// TIA Portal V15.1 export
// export: Created 2024-05-17T05:38:36.3165003Z, ExportSetting WithDefaults, DisplayName Totally Integrated Automation Portal, DisplayVersion V15.1 Update 5, DisplayName TIA Portal Openness, DisplayVersion V15.1 Update 5, DisplayName SINAMICS Startdrive Advanced, DisplayVersion V15.1, DisplayName G130, G150, S120, S150, SINAMICS MV, S210, DisplayVersion V15.1, DisplayName G110M, G120, G120C, G120D, G120P, DisplayVersion V15.1, DisplayName STEP 7 Professional, DisplayVersion V15.1 Update 5, DisplayName STEP 7 Safety, DisplayVersion V15.1, DisplayName WinCC Professional, DisplayVersion V15.1 Update 5, DisplayName SIMATIC Visualization Architect, DisplayVersion V15.1
FUNCTION_BLOCK "LProcPAC-Driver"   // FB1741, SCL
TITLE = LProcPAC-Driver
{ S7_Optimized_Access := 'FALSE' }
AUTHOR : CSTAAL
VERSION : 2.0
// stored: AutoNumber false, IsIECCheckEnabled false, SetENOAutomatically False, UDAEnableTagReadback false
   VAR_INPUT
      ID { ExternalAccessible := 'False'; ExternalVisible := 'False'; ExternalWritable := 'False'} : HW_IO := 0;   // PROFINET = The diagnostic address of the SENTRON PAC; PROFIBUS = The number of the first byte of the input data of the PAC.
      First_Byte_I_O_Data { ExternalAccessible := 'False'; ExternalVisible := 'False'; ExternalWritable := 'False'} : Int := 0;   // The number of the first byte of the control bytes of the SENTRON PAC.
      Connection_Type { ExternalAccessible := 'False'; ExternalVisible := 'False'; ExternalWritable := 'False'} : Int := 1;   // The connection type of the Energy Meter: 1 = single phase, 3 = 3 phase
      Comm_Resource_Limit { ExternalAccessible := 'False'; ExternalVisible := 'False'; ExternalWritable := 'False'} : Int := 4;   // The limit of resources, which can be used by the drviers.
      Automatic_Update { ExternalAccessible := 'False'; ExternalVisible := 'False'; ExternalWritable := 'False'} : Bool := FALSE;   // TRUE = Always update the measurement values as fast as possible.
      Reset_Min_Max { ExternalAccessible := 'False'; ExternalVisible := 'False'; ExternalWritable := 'False'} : Bool := FALSE;   // FALSE ==> TRUE = Reset the minimum and maximum values.
      Reset_Energy_Counter { ExternalAccessible := 'False'; ExternalVisible := 'False'; ExternalWritable := 'False'} : Bool := FALSE;   // FALSE ==> TRUE = Reset the energy counter of the Energy Meter.
      HMI_Bits_Connected { ExternalAccessible := 'False'; ExternalVisible := 'False'; ExternalWritable := 'False'} : Bool := FALSE;   // TRUE = Structure HMI_Bits is connected; FALSE = Structure HMI_Bits is not connected
      Comm_Type { ExternalAccessible := 'False'; ExternalVisible := 'False'; ExternalWritable := 'False'} : Int := 1;   // The communication type, to the SENTRON PAC: 1 = PROFINET, 2 = PROFIBUS
      Min_Max_Calculated { ExternalAccessible := 'False'; ExternalVisible := 'False'; ExternalWritable := 'False'} : Bool := TRUE;   // Only used for PROFIBUS: TRUE = Min-Max-Values are calculated in the driver; FALSE = Min-Max-Values read from the driver.
   END_VAR
   VAR_OUTPUT
      Driver_Control { ExternalAccessible := 'False'; ExternalVisible := 'False'; ExternalWritable := 'False'} : Word;   // Driver Control
      Driver_Data { ExternalAccessible := 'False'; ExternalVisible := 'False'; ExternalWritable := 'False'} : Struct   // The structure including all measurement values. Used for the visualization and the connection to the E2M_Visu block.
         U_L1_L2 { ExternalAccessible := 'False'; ExternalVisible := 'False'; ExternalWritable := 'False'} : Real;
         U_L2_L3 { ExternalAccessible := 'False'; ExternalVisible := 'False'; ExternalWritable := 'False'} : Real;
         U_L3_L1 { ExternalAccessible := 'False'; ExternalVisible := 'False'; ExternalWritable := 'False'} : Real;
         U_L1 { ExternalAccessible := 'False'; ExternalVisible := 'False'; ExternalWritable := 'False'} : Real;
         U_L2 { ExternalAccessible := 'False'; ExternalVisible := 'False'; ExternalWritable := 'False'} : Real;
         U_L3 { ExternalAccessible := 'False'; ExternalVisible := 'False'; ExternalWritable := 'False'} : Real;
         U_L1_L2_min { ExternalAccessible := 'False'; ExternalVisible := 'False'; ExternalWritable := 'False'} : Real;
         U_L2_L3_min { ExternalAccessible := 'False'; ExternalVisible := 'False'; ExternalWritable := 'False'} : Real;
         U_L3_L1_min { ExternalAccessible := 'False'; ExternalVisible := 'False'; ExternalWritable := 'False'} : Real;
         U_L1_min { ExternalAccessible := 'False'; ExternalVisible := 'False'; ExternalWritable := 'False'} : Real;
         U_L2_min { ExternalAccessible := 'False'; ExternalVisible := 'False'; ExternalWritable := 'False'} : Real;
         U_L3_min { ExternalAccessible := 'False'; ExternalVisible := 'False'; ExternalWritable := 'False'} : Real;
         U_L1_L2_max { ExternalAccessible := 'False'; ExternalVisible := 'False'; ExternalWritable := 'False'} : Real;
         U_L2_L3_max { ExternalAccessible := 'False'; ExternalVisible := 'False'; ExternalWritable := 'False'} : Real;
         U_L3_L1_max { ExternalAccessible := 'False'; ExternalVisible := 'False'; ExternalWritable := 'False'} : Real;
         U_L1_max { ExternalAccessible := 'False'; ExternalVisible := 'False'; ExternalWritable := 'False'} : Real;
         U_L2_max { ExternalAccessible := 'False'; ExternalVisible := 'False'; ExternalWritable := 'False'} : Real;
         U_L3_max { ExternalAccessible := 'False'; ExternalVisible := 'False'; ExternalWritable := 'False'} : Real;
         U_PH_PH_Average { ExternalAccessible := 'False'; ExternalVisible := 'False'; ExternalWritable := 'False'} : Real;
         U_PH_N_Average { ExternalAccessible := 'False'; ExternalVisible := 'False'; ExternalWritable := 'False'} : Real;
         U_PH_PH_Average_min { ExternalAccessible := 'False'; ExternalVisible := 'False'; ExternalWritable := 'False'} : Real;
         U_PH_N_Average_min { ExternalAccessible := 'False'; ExternalVisible := 'False'; ExternalWritable := 'False'} : Real;
         U_PH_PH_Average_max { ExternalAccessible := 'False'; ExternalVisible := 'False'; ExternalWritable := 'False'} : Real;
         U_PH_N_Average_max { ExternalAccessible := 'False'; ExternalVisible := 'False'; ExternalWritable := 'False'} : Real;
         I_L1 { ExternalAccessible := 'False'; ExternalVisible := 'False'; ExternalWritable := 'False'} : Real;
         I_L2 { ExternalAccessible := 'False'; ExternalVisible := 'False'; ExternalWritable := 'False'} : Real;
         I_L3 { ExternalAccessible := 'False'; ExternalVisible := 'False'; ExternalWritable := 'False'} : Real;
         I_L1_min { ExternalAccessible := 'False'; ExternalVisible := 'False'; ExternalWritable := 'False'} : Real;
         I_L2_min { ExternalAccessible := 'False'; ExternalVisible := 'False'; ExternalWritable := 'False'} : Real;
         I_L3_min { ExternalAccessible := 'False'; ExternalVisible := 'False'; ExternalWritable := 'False'} : Real;
         I_L1_max { ExternalAccessible := 'False'; ExternalVisible := 'False'; ExternalWritable := 'False'} : Real;
         I_L2_max { ExternalAccessible := 'False'; ExternalVisible := 'False'; ExternalWritable := 'False'} : Real;
         I_L3_max { ExternalAccessible := 'False'; ExternalVisible := 'False'; ExternalWritable := 'False'} : Real;
         I_Average { ExternalAccessible := 'False'; ExternalVisible := 'False'; ExternalWritable := 'False'} : Real;
         I_Average_min { ExternalAccessible := 'False'; ExternalVisible := 'False'; ExternalWritable := 'False'} : Real;
         I_Average_max { ExternalAccessible := 'False'; ExternalVisible := 'False'; ExternalWritable := 'False'} : Real;
         f { ExternalAccessible := 'False'; ExternalVisible := 'False'; ExternalWritable := 'False'} : Real;
         f_min { ExternalAccessible := 'False'; ExternalVisible := 'False'; ExternalWritable := 'False'} : Real;
         f_max { ExternalAccessible := 'False'; ExternalVisible := 'False'; ExternalWritable := 'False'} : Real;
         S_Total { ExternalAccessible := 'False'; ExternalVisible := 'False'; ExternalWritable := 'False'} : Real;
         S_Total_min { ExternalAccessible := 'False'; ExternalVisible := 'False'; ExternalWritable := 'False'} : Real;
         S_Total_max { ExternalAccessible := 'False'; ExternalVisible := 'False'; ExternalWritable := 'False'} : Real;
         P_Total { ExternalAccessible := 'False'; ExternalVisible := 'False'; ExternalWritable := 'False'} : Real;
         P_Total_min { ExternalAccessible := 'False'; ExternalVisible := 'False'; ExternalWritable := 'False'} : Real;
         P_Total_max { ExternalAccessible := 'False'; ExternalVisible := 'False'; ExternalWritable := 'False'} : Real;
         Q_Total { ExternalAccessible := 'False'; ExternalVisible := 'False'; ExternalWritable := 'False'} : Real;
         Q_Total_min { ExternalAccessible := 'False'; ExternalVisible := 'False'; ExternalWritable := 'False'} : Real;
         Q_Total_max { ExternalAccessible := 'False'; ExternalVisible := 'False'; ExternalWritable := 'False'} : Real;
         Cos_L1 { ExternalAccessible := 'False'; ExternalVisible := 'False'; ExternalWritable := 'False'} : Real;
         Cos_L1_min { ExternalAccessible := 'False'; ExternalVisible := 'False'; ExternalWritable := 'False'} : Real;
         Cos_L1_max { ExternalAccessible := 'False'; ExternalVisible := 'False'; ExternalWritable := 'False'} : Real;
         Cos_L2 { ExternalAccessible := 'False'; ExternalVisible := 'False'; ExternalWritable := 'False'} : Real;
         Cos_L2_min { ExternalAccessible := 'False'; ExternalVisible := 'False'; ExternalWritable := 'False'} : Real;
         Cos_L2_max { ExternalAccessible := 'False'; ExternalVisible := 'False'; ExternalWritable := 'False'} : Real;
         Cos_L3 { ExternalAccessible := 'False'; ExternalVisible := 'False'; ExternalWritable := 'False'} : Real;
         Cos_L3_min { ExternalAccessible := 'False'; ExternalVisible := 'False'; ExternalWritable := 'False'} : Real;
         Cos_L3_max { ExternalAccessible := 'False'; ExternalVisible := 'False'; ExternalWritable := 'False'} : Real;
         Cos_Total { ExternalAccessible := 'False'; ExternalVisible := 'False'; ExternalWritable := 'False'} : Real;
         Cos_Total_min { ExternalAccessible := 'False'; ExternalVisible := 'False'; ExternalWritable := 'False'} : Real;
         Cos_Total_max { ExternalAccessible := 'False'; ExternalVisible := 'False'; ExternalWritable := 'False'} : Real;
         S_L1 { ExternalAccessible := 'False'; ExternalVisible := 'False'; ExternalWritable := 'False'} : Real;
         S_L2 { ExternalAccessible := 'False'; ExternalVisible := 'False'; ExternalWritable := 'False'} : Real;
         S_L3 { ExternalAccessible := 'False'; ExternalVisible := 'False'; ExternalWritable := 'False'} : Real;
         S_L1_min { ExternalAccessible := 'False'; ExternalVisible := 'False'; ExternalWritable := 'False'} : Real;
         S_L2_min { ExternalAccessible := 'False'; ExternalVisible := 'False'; ExternalWritable := 'False'} : Real;
         S_L3_min { ExternalAccessible := 'False'; ExternalVisible := 'False'; ExternalWritable := 'False'} : Real;
         S_L1_max { ExternalAccessible := 'False'; ExternalVisible := 'False'; ExternalWritable := 'False'} : Real;
         S_L2_max { ExternalAccessible := 'False'; ExternalVisible := 'False'; ExternalWritable := 'False'} : Real;
         S_L3_max { ExternalAccessible := 'False'; ExternalVisible := 'False'; ExternalWritable := 'False'} : Real;
         P_L1 { ExternalAccessible := 'False'; ExternalVisible := 'False'; ExternalWritable := 'False'} : Real;
         P_L2 { ExternalAccessible := 'False'; ExternalVisible := 'False'; ExternalWritable := 'False'} : Real;
         P_L3 { ExternalAccessible := 'False'; ExternalVisible := 'False'; ExternalWritable := 'False'} : Real;
         P_L1_min { ExternalAccessible := 'False'; ExternalVisible := 'False'; ExternalWritable := 'False'} : Real;
         P_L2_min { ExternalAccessible := 'False'; ExternalVisible := 'False'; ExternalWritable := 'False'} : Real;
         P_L3_min { ExternalAccessible := 'False'; ExternalVisible := 'False'; ExternalWritable := 'False'} : Real;
         P_L1_max { ExternalAccessible := 'False'; ExternalVisible := 'False'; ExternalWritable := 'False'} : Real;
         P_L2_max { ExternalAccessible := 'False'; ExternalVisible := 'False'; ExternalWritable := 'False'} : Real;
         P_L3_max { ExternalAccessible := 'False'; ExternalVisible := 'False'; ExternalWritable := 'False'} : Real;
         Q_L1 { ExternalAccessible := 'False'; ExternalVisible := 'False'; ExternalWritable := 'False'} : Real;
         Q_L2 { ExternalAccessible := 'False'; ExternalVisible := 'False'; ExternalWritable := 'False'} : Real;
         Q_L3 { ExternalAccessible := 'False'; ExternalVisible := 'False'; ExternalWritable := 'False'} : Real;
         Q_L1_min { ExternalAccessible := 'False'; ExternalVisible := 'False'; ExternalWritable := 'False'} : Real;
         Q_L2_min { ExternalAccessible := 'False'; ExternalVisible := 'False'; ExternalWritable := 'False'} : Real;
         Q_L3_min { ExternalAccessible := 'False'; ExternalVisible := 'False'; ExternalWritable := 'False'} : Real;
         Q_L1_max { ExternalAccessible := 'False'; ExternalVisible := 'False'; ExternalWritable := 'False'} : Real;
         Q_L2_max { ExternalAccessible := 'False'; ExternalVisible := 'False'; ExternalWritable := 'False'} : Real;
         Q_L3_max { ExternalAccessible := 'False'; ExternalVisible := 'False'; ExternalWritable := 'False'} : Real;
         E_Active_Rate1_Import { ExternalAccessible := 'False'; ExternalVisible := 'False'; ExternalWritable := 'False'} : Real;
         E_Active_Rate2_Import { ExternalAccessible := 'False'; ExternalVisible := 'False'; ExternalWritable := 'False'} : Real;
         E_Active_Rate1_Export { ExternalAccessible := 'False'; ExternalVisible := 'False'; ExternalWritable := 'False'} : Real;
         E_Active_Rate2_Export { ExternalAccessible := 'False'; ExternalVisible := 'False'; ExternalWritable := 'False'} : Real;
         E_Reactive_Rate1_Import { ExternalAccessible := 'False'; ExternalVisible := 'False'; ExternalWritable := 'False'} : Real;
         E_Reactive_Rate2_Import { ExternalAccessible := 'False'; ExternalVisible := 'False'; ExternalWritable := 'False'} : Real;
         E_Reactive_Rate1_Export { ExternalAccessible := 'False'; ExternalVisible := 'False'; ExternalWritable := 'False'} : Real;
         E_Reactive_Rate2_Export { ExternalAccessible := 'False'; ExternalVisible := 'False'; ExternalWritable := 'False'} : Real;
         E_Apparent_Rate1_Import { ExternalAccessible := 'False'; ExternalVisible := 'False'; ExternalWritable := 'False'} : Real;
         E_Apparent_Rate2_Import { ExternalAccessible := 'False'; ExternalVisible := 'False'; ExternalWritable := 'False'} : Real;
         RTime_Data_Energy { ExternalAccessible := 'False'; ExternalVisible := 'False'; ExternalWritable := 'False'} : Date_And_Time;
         RTime_Data_Value { ExternalAccessible := 'False'; ExternalVisible := 'False'; ExternalWritable := 'False'} : Date_And_Time;
         U_PH_PH_Mod { ExternalAccessible := 'False'; ExternalVisible := 'False'; ExternalWritable := 'False'} : Word;
         U_PH_N_Mod { ExternalAccessible := 'False'; ExternalVisible := 'False'; ExternalWritable := 'False'} : Word;
         I_Mod { ExternalAccessible := 'False'; ExternalVisible := 'False'; ExternalWritable := 'False'} : Word;
         S_Mod { ExternalAccessible := 'False'; ExternalVisible := 'False'; ExternalWritable := 'False'} : Word;
         P_Mod { ExternalAccessible := 'False'; ExternalVisible := 'False'; ExternalWritable := 'False'} : Word;
         Q_Mod { ExternalAccessible := 'False'; ExternalVisible := 'False'; ExternalWritable := 'False'} : Word;
         E_Mod { ExternalAccessible := 'False'; ExternalVisible := 'False'; ExternalWritable := 'False'} : Word;
         f_Mod { ExternalAccessible := 'False'; ExternalVisible := 'False'; ExternalWritable := 'False'} : Word;
         Cos_Mod { ExternalAccessible := 'False'; ExternalVisible := 'False'; ExternalWritable := 'False'} : Word;
         Calculate_Value1 { ExternalAccessible := 'False'; ExternalVisible := 'False'; ExternalWritable := 'False'} : Word;
         Calculate_Value2 { ExternalAccessible := 'False'; ExternalVisible := 'False'; ExternalWritable := 'False'} : Word;
         Calculate_Value3 { ExternalAccessible := 'False'; ExternalVisible := 'False'; ExternalWritable := 'False'} : Word;
         Calculate_Value4 { ExternalAccessible := 'False'; ExternalVisible := 'False'; ExternalWritable := 'False'} : Word;
         Calculate_Value5 { ExternalAccessible := 'False'; ExternalVisible := 'False'; ExternalWritable := 'False'} : Word;
         Calculate_Value6 { ExternalAccessible := 'False'; ExternalVisible := 'False'; ExternalWritable := 'False'} : Word;
         Energy_Meter_Unit { ExternalAccessible := 'False'; ExternalVisible := 'False'; ExternalWritable := 'False'} : Word;
         Rest_Start_Auto { ExternalAccessible := 'False'; ExternalVisible := 'False'; ExternalWritable := 'False'} : Bool;
         Read_Value { ExternalAccessible := 'False'; ExternalVisible := 'False'; ExternalWritable := 'False'} : Bool;
         Connection_Type { ExternalAccessible := 'False'; ExternalVisible := 'False'; ExternalWritable := 'False'} : Int;
         Driver_Error { ExternalAccessible := 'False'; ExternalVisible := 'False'; ExternalWritable := 'False'} : Int;
      END_STRUCT;
      Energy_Counter { ExternalAccessible := 'False'; ExternalVisible := 'False'; ExternalWritable := 'False'} : Struct   // The structure with all energy counter as 64-Bit float values.
         Active_Rate1_Imp_Raw { ExternalAccessible := 'False'; ExternalVisible := 'False'; ExternalWritable := 'False'} : DInt;
         Active_Rate1_Imp_Fine { ExternalAccessible := 'False'; ExternalVisible := 'False'; ExternalWritable := 'False'} : DInt;
         Active_Rate1_Exp_Raw { ExternalAccessible := 'False'; ExternalVisible := 'False'; ExternalWritable := 'False'} : DInt;
         Active_Rate1_Exp_Fine { ExternalAccessible := 'False'; ExternalVisible := 'False'; ExternalWritable := 'False'} : DInt;
         Active_Rate2_Imp_Raw { ExternalAccessible := 'False'; ExternalVisible := 'False'; ExternalWritable := 'False'} : DInt;
         Active_Rate2_Imp_Fine { ExternalAccessible := 'False'; ExternalVisible := 'False'; ExternalWritable := 'False'} : DInt;
         Active_Rate2_Exp_Raw { ExternalAccessible := 'False'; ExternalVisible := 'False'; ExternalWritable := 'False'} : DInt;
         Active_Rate2_Exp_Fine { ExternalAccessible := 'False'; ExternalVisible := 'False'; ExternalWritable := 'False'} : DInt;
         Reactive_Rate1_Imp_Raw { ExternalAccessible := 'False'; ExternalVisible := 'False'; ExternalWritable := 'False'} : DInt;
         Reactive_Rate1_Imp_Fine { ExternalAccessible := 'False'; ExternalVisible := 'False'; ExternalWritable := 'False'} : DInt;
         Reactive_Rate1_Exp_Raw { ExternalAccessible := 'False'; ExternalVisible := 'False'; ExternalWritable := 'False'} : DInt;
         Reactive_Rate1_Exp_Fine { ExternalAccessible := 'False'; ExternalVisible := 'False'; ExternalWritable := 'False'} : DInt;
         Reactive_Rate2_Imp_Raw { ExternalAccessible := 'False'; ExternalVisible := 'False'; ExternalWritable := 'False'} : DInt;
         Reactive_Rate2_Imp_Fine { ExternalAccessible := 'False'; ExternalVisible := 'False'; ExternalWritable := 'False'} : DInt;
         Reactive_Rate2_Exp_Raw { ExternalAccessible := 'False'; ExternalVisible := 'False'; ExternalWritable := 'False'} : DInt;
         Reactive_Rate2_Exp_Fine { ExternalAccessible := 'False'; ExternalVisible := 'False'; ExternalWritable := 'False'} : DInt;
         Apparent_Rate1_Imp_Raw { ExternalAccessible := 'False'; ExternalVisible := 'False'; ExternalWritable := 'False'} : DInt;
         Apparent_Rate1_Imp_Fine { ExternalAccessible := 'False'; ExternalVisible := 'False'; ExternalWritable := 'False'} : DInt;
         Apparent_Rate2_Imp_Raw { ExternalAccessible := 'False'; ExternalVisible := 'False'; ExternalWritable := 'False'} : DInt;
         Apparent_Rate2_Imp_Fine { ExternalAccessible := 'False'; ExternalVisible := 'False'; ExternalWritable := 'False'} : DInt;
      END_STRUCT;
      Time_Between_Update { ExternalAccessible := 'False'; ExternalVisible := 'False'; ExternalWritable := 'False'} : Time := T#0MS;   // The time between the current and the last update of the measurement values.
      Time_Between_Update_Max { ExternalAccessible := 'False'; ExternalVisible := 'False'; ExternalWritable := 'False'} : Time := T#0MS;   // The maximum time between two measurement value updates.
      Time_Stamp_Meas_Values { ExternalAccessible := 'False'; ExternalVisible := 'False'; ExternalWritable := 'False'} : Date_And_Time := DT#1990-01-01-00:00:00;   // The time stamp of the currently available measurement values.
      Error_Location { ExternalAccessible := 'False'; ExternalVisible := 'False'; ExternalWritable := 'False'} : Word := WORD#16#0000;   // The error location or the status of the block. Detailed information in the manual.
      Error_Code { ExternalAccessible := 'False'; ExternalVisible := 'False'; ExternalWritable := 'False'} : DWord := DWORD#16#0000_0000;   // The error code in case of an error of the block, otherwise 0. Detailed information in the manual.
   END_VAR
   VAR_IN_OUT
      HMI_Bits : Struct   // The structure with the feedback of the HMI. Used for the visualization and the connection to the E2M_Visu block.
         Start_Acyclic : Bool;
         Start_Auto : Bool;
         Reset_min_max_Data : Bool;
         Reset_Energy_Meter : Bool;
      END_STRUCT;
      Comm_Resource_Counter { ExternalAccessible := 'False'; ExternalVisible := 'False'; ExternalWritable := 'False'} : Int := 0;   // The counter of the currently used resources from all E2M drivers.
   END_VAR
   VAR
      Read_Data_Record { ExternalAccessible := 'False'; ExternalVisible := 'False'; ExternalWritable := 'False'; S7_SetPoint := 'True'} : RDREC;
      Write_Data_Record { ExternalAccessible := 'False'; ExternalVisible := 'False'; ExternalWritable := 'False'; S7_SetPoint := 'True'} : WRREC;
   END_VAR
   VAR DB_SPECIFIC
      Time_Measurement { ExternalAccessible := 'False'; ExternalVisible := 'False'; ExternalWritable := 'False'; S7_SetPoint := 'True'} : TON_TIME;
      Error_Retry_Timer { ExternalAccessible := 'False'; ExternalVisible := 'False'; ExternalWritable := 'False'; S7_SetPoint := 'True'} : TON_TIME;
      Watchdog { ExternalAccessible := 'False'; ExternalVisible := 'False'; ExternalWritable := 'False'; S7_SetPoint := 'True'} : TON_TIME;
      Reset_Timer { ExternalAccessible := 'False'; ExternalVisible := 'False'; ExternalWritable := 'False'; S7_SetPoint := 'True'} : TON_TIME;
   END_VAR
   VAR
      LREAL_TO_DINT { ExternalAccessible := 'False'; ExternalVisible := 'False'; ExternalWritable := 'False'; S7_SetPoint := 'True'} : "LProcPAC-Conversion";
   END_VAR
   VAR DB_SPECIFIC
      Input_Variables_OK { ExternalAccessible := 'False'; ExternalVisible := 'False'; ExternalWritable := 'False'} : Bool := FALSE;
      HMI_Input_Bits_Connected { ExternalAccessible := 'False'; ExternalVisible := 'False'; ExternalWritable := 'False'} : Bool := FALSE;
      Reset_En_Count_Request { ExternalAccessible := 'False'; ExternalVisible := 'False'; ExternalWritable := 'False'} : Bool := FALSE;
      Reset_Min_Max_Request { ExternalAccessible := 'False'; ExternalVisible := 'False'; ExternalWritable := 'False'} : Bool := FALSE;
      Read_Data_Rec_Request { ExternalAccessible := 'False'; ExternalVisible := 'False'; ExternalWritable := 'False'} : Bool := FALSE;
      Write_Data_Rec_Request { ExternalAccessible := 'False'; ExternalVisible := 'False'; ExternalWritable := 'False'} : Bool := FALSE;
      Start_Acyclic_HMI_Old { ExternalAccessible := 'False'; ExternalVisible := 'False'; ExternalWritable := 'False'} : Bool := FALSE;
      Reset_Energy_HMI_Old { ExternalAccessible := 'False'; ExternalVisible := 'False'; ExternalWritable := 'False'} : Bool := FALSE;
      Reset_Energy_Old { ExternalAccessible := 'False'; ExternalVisible := 'False'; ExternalWritable := 'False'} : Bool := FALSE;
      Reset_Min_Max_HMI_Old { ExternalAccessible := 'False'; ExternalVisible := 'False'; ExternalWritable := 'False'} : Bool := FALSE;
      Reset_Min_Max_Old { ExternalAccessible := 'False'; ExternalVisible := 'False'; ExternalWritable := 'False'} : Bool := FALSE;
      Error_Retry_Timer_Run { ExternalAccessible := 'False'; ExternalVisible := 'False'; ExternalWritable := 'False'} : Bool := FALSE;
      Watchdog_Run { ExternalAccessible := 'False'; ExternalVisible := 'False'; ExternalWritable := 'False'} : Bool := FALSE;
      Reset_Timer_Run { ExternalAccessible := 'False'; ExternalVisible := 'False'; ExternalWritable := 'False'} : Bool := FALSE;
      PE_Request_Reference { ExternalAccessible := 'False'; ExternalVisible := 'False'; ExternalWritable := 'False'} : Byte := BYTE#16#01;
      Sm_State { ExternalAccessible := 'False'; ExternalVisible := 'False'; ExternalWritable := 'False'} : Int := 0;
      Sm_State_Next { ExternalAccessible := 'False'; ExternalVisible := 'False'; ExternalWritable := 'False'} : Int := 0;
      Rd_Rec_Index { ExternalAccessible := 'False'; ExternalVisible := 'False'; ExternalWritable := 'False'} : Int := 0;
      Rd_Rec_Max_Length { ExternalAccessible := 'False'; ExternalVisible := 'False'; ExternalWritable := 'False'} : Int := 0;
      Wr_Rec_Index { ExternalAccessible := 'False'; ExternalVisible := 'False'; ExternalWritable := 'False'} : Int := 0;
      Wr_Rec_Max_Length { ExternalAccessible := 'False'; ExternalVisible := 'False'; ExternalWritable := 'False'} : Int := 0;
      Error_Retry_Counter { ExternalAccessible := 'False'; ExternalVisible := 'False'; ExternalWritable := 'False'} : Int := 0;
      Time_to_update { ExternalAccessible := 'False'; ExternalVisible := 'False'; ExternalWritable := 'False'} : Time := T#0MS;
      HMI_Bits_Internal { ExternalAccessible := 'False'; ExternalVisible := 'False'; ExternalWritable := 'False'} : Struct
         Start_Acyclic { ExternalAccessible := 'False'; ExternalVisible := 'False'; ExternalWritable := 'False'} : Bool := FALSE;
         Start_Auto { ExternalAccessible := 'False'; ExternalVisible := 'False'; ExternalWritable := 'False'} : Bool := FALSE;
         Reset_min_max_Data { ExternalAccessible := 'False'; ExternalVisible := 'False'; ExternalWritable := 'False'} : Bool := FALSE;
         Reset_Energy_Meter { ExternalAccessible := 'False'; ExternalVisible := 'False'; ExternalWritable := 'False'} : Bool := FALSE;
      END_STRUCT;
      Receive_Data_Buffer { ExternalAccessible := 'False'; ExternalVisible := 'False'; ExternalWritable := 'False'} : Array[1..1002] of Byte;
   END_VAR
   VAR
      V_PN_Meas_Data_Res_1 AT Receive_Data_Buffer : Struct   // AT Receive_Data_Buffer : Struct
         Block_Header : Struct
            Block_Type : Word;
            Block_Length : Int;
            Block_Version : Word;
         END_STRUCT;
         Response_Header : Struct
            Service_Request_ID : Byte;
            Request_Reference : Byte;
         END_STRUCT;
         Service_Header_Response : Struct
            Status : Byte;
            Data_Struct_Identifier : Byte;
         END_STRUCT;
         Service_Data_Response : Struct
            Count_Meas_Values : Byte;
            Reserver : Byte;
            Meas_Values_32Bit : Array[1..50] of Struct
               Length_Of_Struct : Int;
               Meas_Data_Struct : Byte;
               Meas_ID_HB : Byte;
               Meas_ID_LB : Byte;
               Meas_Status : Byte;
               Meas_Value : Real;
            END_STRUCT;
         END_STRUCT;
      END_STRUCT;
      V_DP_Meas_Data_Res AT Receive_Data_Buffer : Struct   // AT Receive_Data_Buffer : Struct
         U_L1 : Real;
         U_L2 : Real;
         U_L3 : Real;
         U_L1_L2 : Real;
         U_L2_L3 : Real;
         U_L3_L1 : Real;
         I_L1 : Real;
         I_L2 : Real;
         I_L3 : Real;
         S_L1 : Real;
         S_L2 : Real;
         S_L3 : Real;
         P_L1 : Real;
         P_L2 : Real;
         P_L3 : Real;
         Q_L1 : Real;
         Q_L2 : Real;
         Q_L3 : Real;
         Cos_L1 : Real;
         Cos_L2 : Real;
         Cos_L3 : Real;
         f : Real;
         U_PH_N_Average : Real;
         U_PH_PH_Average : Real;
         I_Average : Real;
         S_Total : Real;
         P_Total : Real;
         Q_Total : Real;
         Cos_Total : Real;
         E_Active_Rate1_Im_HW : DWord;
         E_Active_Rate1_Im_LW : DWord;
         E_Active_Rate2_Im_HW : DWord;
         E_Active_Rate2_Im_LW : DWord;
         E_Active_Rate1_Ex_HW : DWord;
         E_Active_Rate1_Ex_LW : DWord;
         E_Active_Rate2_Ex_HW : DWord;
         E_Active_Rate2_Ex_LW : DWord;
         E_Reactive_Rate1_Im_HW : DWord;
         E_Reactive_Rate1_Im_LW : DWord;
         E_Reactive_Rate2_Im_HW : DWord;
         E_Reactive_Rate2_Im_LW : DWord;
         E_Reactive_Rate1_Ex_HW : DWord;
         E_Reactive_Rate1_Ex_LW : DWord;
         E_Reactive_Rate2_Ex_HW : DWord;
         E_Reactive_Rate2_Ex_LW : DWord;
         E_Apparent_Rate1_Im_HW : DWord;
         E_Apparent_Rate1_Im_LW : DWord;
         E_Apparent_Rate2_Im_HW : DWord;
         E_Apparent_Rate2_Im_LW : DWord;
      END_STRUCT;
      V_DP_Meas_Reset AT Receive_Data_Buffer : Struct   // AT Receive_Data_Buffer : Struct
         Meas_Values : Array[1..47] of DWord;
      END_STRUCT;
      V_DP_Meas_Min_Max AT Receive_Data_Buffer : Struct   // AT Receive_Data_Buffer : Struct
         U_L1_Max : Real;
         U_L2_Max : Real;
         U_L3_Max : Real;
         U_L1_L2_Max : Real;
         U_L2_L3_Max : Real;
         U_L3_L1_Max : Real;
         I_L1_Max : Real;
         I_L2_Max : Real;
         I_L3_Max : Real;
         S_L1_Max : Real;
         S_L2_Max : Real;
         S_L3_Max : Real;
         P_L1_Max : Real;
         P_L2_Max : Real;
         P_L3_Max : Real;
         Q_L1_Max : Real;
         Q_L2_Max : Real;
         Q_L3_Max : Real;
         Cos_L1_Max : Real;
         Cos_L2_Max : Real;
         Cos_L3_Max : Real;
         f_Max : Real;
         U_PH_N_Average_Max : Real;
         U_PH_PH_Average_Max : Real;
         I_Average_Max : Real;
         S_Total_Max : Real;
         P_Total_Max : Real;
         Q_Total_Max : Real;
         Cos_Total_Max : Real;
         U_L1_Min : Real;
         U_L2_Min : Real;
         U_L3_Min : Real;
         U_L1_L2_Min : Real;
         U_L2_L3_Min : Real;
         U_L3_L1_Min : Real;
         I_L1_Min : Real;
         I_L2_Min : Real;
         I_L3_Min : Real;
         S_L1_Min : Real;
         S_L2_Min : Real;
         S_L3_Min : Real;
         P_L1_Min : Real;
         P_L2_Min : Real;
         P_L3_Min : Real;
         Q_L1_Min : Real;
         Q_L2_Min : Real;
         Q_L3_Min : Real;
         Cos_L1_Min : Real;
         Cos_L2_Min : Real;
         Cos_L3_Min : Real;
         f_Min : Real;
         U_PH_N_Average_Min : Real;
         U_PH_PH_Average_Min : Real;
         I_Average_Min : Real;
         S_Total_Min : Real;
         P_Total_Min : Real;
         Q_Total_Min : Real;
         Cos_Total_Min : Real;
      END_STRUCT;
      V_DP_Min_Max_Reset AT Receive_Data_Buffer : Struct   // AT Receive_Data_Buffer : Struct
         Meas_Values : Array[1..58] of DWord;
      END_STRUCT;
      V_PN_Meas_Data_Res_2 AT Receive_Data_Buffer : Struct   // AT Receive_Data_Buffer : Struct
         Block_Header : Struct
            Block_Type : Word;
            Block_Length : Int;
            Block_Version : Word;
         END_STRUCT;
         Response_Header : Struct
            Service_Request_ID : Byte;
            Request_Reference : Byte;
         END_STRUCT;
         Service_Header_Response : Struct
            Status : Byte;
            Data_Struct_Identifier : Byte;
         END_STRUCT;
         Service_Data_Response : Struct
            Count_Meas_Values : Byte;
            Reserver : Byte;
            Meas_Values_32Bit : Array[51..87] of Struct
               Length_Of_Struct : Int;
               Meas_Data_Struct : Byte;
               Meas_ID_HB : Byte;
               Meas_ID_LB : Byte;
               Meas_Status : Byte;
               Meas_Value : Real;
            END_STRUCT;
            Meas_Values_64Bit : Array[88..92] of Struct
               Length_Of_Struct : Int;
               Meas_Data_Struct : Byte;
               Meas_ID_HB : Byte;
               Meas_ID_LB : Byte;
               Meas_Status : Byte;
               Meas_Value_H : DWord;
               Meas_Value_L : DWord;
            END_STRUCT;
         END_STRUCT;
      END_STRUCT;
   END_VAR
   VAR DB_SPECIFIC
      Send_Data_Buffer { ExternalAccessible := 'False'; ExternalVisible := 'False'; ExternalWritable := 'False'} : Array[1..240] of Byte;
   END_VAR
   VAR
      V_PN_Measurement_Data_1 AT Send_Data_Buffer : Struct   // AT Send_Data_Buffer : Struct
         Block_Header : Struct
            Block_Type : Word;
            Block_Length : Int;
            Block_Version : Word;
         END_STRUCT;
         Request_Header : Struct
            Service_Request_ID : Byte;
            Request_Reference : Byte;
         END_STRUCT;
         Service_Header_Request : Struct
            Modifier : Byte;
            Data_Struct_Identifier : Byte;
         END_STRUCT;
         Service_Data_Request : Struct
            Count_Meas_Values : Byte;
            Reserver : Byte;
            Meas_Values : Array[1..50] of Int;
         END_STRUCT;
      END_STRUCT;
      V_DP_Measurement_Data AT Send_Data_Buffer : Struct   // AT Send_Data_Buffer : Struct
         Measurement_Data : Array[1..58] of Struct
            Measurement_ID : Int;
            Measurement_Len : Int;
         END_STRUCT;
      END_STRUCT;
      V_DP_ResetData AT Send_Data_Buffer : Struct   // AT Send_Data_Buffer : Struct
         Command_ID : Array[1..2] of Struct
            Command_ID : Int;
            Command_Len : Int;
            Command_Value : Int;
         END_STRUCT;
      END_STRUCT;
      V_PN_Measurement_Data_2 AT Send_Data_Buffer : Struct   // AT Send_Data_Buffer : Struct
         Block_Header : Struct
            Block_Type : Word;
            Block_Length : Int;
            Block_Version : Word;
         END_STRUCT;
         Request_Header : Struct
            Service_Request_ID : Byte;
            Request_Reference : Byte;
         END_STRUCT;
         Service_Header_Request : Struct
            Modifier : Byte;
            Data_Struct_Identifier : Byte;
         END_STRUCT;
         Service_Data_Request : Struct
            Count_Meas_Values : Byte;
            Reserver : Byte;
            Meas_Values : Array[51..92] of Int;
         END_STRUCT;
      END_STRUCT;
   END_VAR
   VAR_TEMP
      General_Ret_Val : Int;
      Index : Int;
      In_Out_Pointer_Check : Any;
      VIn_Out_Pointer_Check AT In_Out_Pointer_Check : Struct   // AT In_Out_Pointer_Check : Struct
         ID_Type : Word;
         Count : Word;
         DB_Number : Word;
         DB_Offset : DWord;
      END_STRUCT;
   END_VAR
   VAR CONSTANT
      CONNECTION_SINGLE_PHASE : Int := 1;
      CONNECTION_THREE_PHASE : Int := 3;
      PROFINET : Int := 1;
      PROFIBUS : Int := 2;
      RECORD_47_FLEX_ACCESS_MEASUREMENT_INDEX : Int := 47;
      RECORD_PROFIENERGY_INDEX : Word := WORD#16#80A0;
      RECORD_47_WRITE_MEASUREMENT_VALUES_LENGTH : Int := 12;
      RECORD_47_READ_MEASUREMENT_VALUES_LENGTH : Int := 196;
      RECORD_47_WRITE_MINMAX_LEN : Int := 8;
      RECORD_47_READ_MIN_MAX_VALUES_LENGTH : Int := 232;
      RECORD_PE_WRITE_LEN_1 : Int := 112;
      RECORD_PE_WRITE_LEN_2 : Int := 96;
      RECORD_PE_READ_LEN_1 : Int := 512;
      RECORD_PE_READ_LEN_2 : Int := 452;
      RECORD_PE_COUNT_MEAS_1 : Int := 50;
      RECORD_PE_COUNT_MEAS_2 : Int := 42;
      DP_CMD_RESET_MINIMUM_VALUES : Word := WORD#16#EA63;
      DP_CMD_RESET_MAXIMUM_VALUES : Word := WORD#16#EA62;
      DP_CMD_RESET_ENERGY_COUNTER : Word := WORD#16#EA64;
      ERR_LOC_WRITE_MEAS_1 : Word := WORD#16#1311;
      ERR_LOC_WRITE_MEAS_2 : Word := WORD#16#1312;
      ERR_LOC_WRITE_MIN_MAX_VALUES : Word := WORD#16#1313;
      ERR_LOC_WRITE_RES_MIN_MAX : Word := WORD#16#1314;
      ERR_LOC_WRITE_RESET_ENERGY_COUNTER : Word := WORD#16#1315;
      ERR_LOC_READ_MEAS_1 : Word := WORD#16#1321;
      ERR_LOC_READ_MEAS_2 : Word := WORD#16#1322;
      ERR_LOC_READ_MIN_MAX_VALUES : Word := WORD#16#1323;
      ERR_LOC_INVALID_ID : Word := WORD#16#1371;
      ERR_LOC_INVALID_CONNECTION_TYPE : Word := WORD#16#1372;
      ERR_LOC_INVALID_COMM_LIMIT : Word := WORD#16#1373;
      ERR_LOC_INVALID_IO_BYTE : Word := WORD#16#1374;
      ERR_LOC_INVALID_BACKUP_TIME : Word := WORD#16#1375;
      ERR_LOC_INVALID_COMM_COUNTER : Word := WORD#16#1376;
      ERR_LOC_INVALID_COMM_TYPE : Word := WORD#16#1377;
      ERR_LOC_NO_POWER : Word := WORD#16#1381;
      ERR_LOC_PN_INV_BLOCK_1 : Word := WORD#16#1390;
      ERR_LOC_PN_INV_REQ_ID_1 : Word := WORD#16#1391;
      ERR_LOC_PN_INV_REQ_REF_1 : Word := WORD#16#1392;
      ERR_LOC_PN_PE_CMD_FAIL_1 : Word := WORD#16#1393;
      ERR_LOC_PN_INV_DATSTR_1 : Word := WORD#16#1394;
      ERR_LOC_PN_INV_BLOCK_2 : Word := WORD#16#1395;
      ERR_LOC_PN_INVALID_REQUEST_ID_2 : Word := WORD#16#1396;
      ERR_LOC_PN_INV_REQ_REF_2 : Word := WORD#16#1397;
      ERR_LOC_PN_PE_CMD_FAIL_2 : Word := WORD#16#1398;
      ERR_LOC_PN_INV_DATSTR_2 : Word := WORD#16#1399;
      STATUS_IDLE : Word := WORD#16#0000;
      STATUS_WAIT_FOR_RESOURCE : Word := WORD#16#7001;
      STATUS_READ_MEAS : Word := WORD#16#7002;
      STATUS_RESET_MIN_MAX_VALUES : Word := WORD#16#7003;
      STATUS_RESET_ENERGY_COUNTER : Word := WORD#16#7004;
      ERROR_CODE_DEVICE_BUSY : DWord := DWORD#16#DE80_C200;
      ERR_CODE_GENERAL : DWord := DWORD#16#0000_0001;
      ERROR_RETRY_LIMIT : Int := 10;
      DATA_TYPE_WORD : Word := WORD#16#1004;
      DATA_TYPE_INT : Word := WORD#16#1005;
      PN_BLOCK_TYPE_READ : Word := WORD#16#0801;
      PN_REQUEST_ID_GET_MEASUREMENT_VALUES : Byte := BYTE#16#10;
      BIT_RESET_ENERGY_COUNTER : Int := 2;
      BIT_RESET_MINIMUM_VALUES : Int := 0;
      BIT_RESET_MAXIMUM_VALUES : Int := 1;
      TIME_WATCHDOG : Time := T#2S;
      TIME_RETRY_TIMER : Time := T#100MS;
      TIME_RESET_TIMER : Time := T#1S;
      SM_IDLE : Int := 0;
      SM_MEAS_WAIT_RESOURCE : Int := 11;
      SM_WRITE_MEAS_WAIT_RESP : Int := 12;
      SM_READ_MEAS_WAIT_RESP : Int := 13;
      SM_READ_MEAS_WAIT_TIME : Int := 14;
      SM_WRITE_MEAS_PN_WAIT_RESP : Int := 15;
      SM_READ_MEAS_PN_WAIT_RESP : Int := 16;
      SM_READ_MEAS_PN_WAIT_TIME : Int := 17;
      SM_WRITE_MINMAX_WAIT_RESP : Int := 18;
      SM_READ_MINMAX_WAIT_RESP : Int := 19;
      SM_WRITE_MINMAX_DP_RESP : Int := 24;
      SM_READ_MINMAX_DP_WAIT_RESP : Int := 25;
      PE_ID_U_L1 : Int := 1;
      PE_ID_U_L2 : Int := 2;
      PE_ID_U_L3 : Int := 3;
      PE_ID_U_L1_L2 : Int := 4;
      PE_ID_U_L2_L3 : Int := 5;
      PE_ID_U_L3_L1 : Int := 6;
      PE_ID_I_L1 : Int := 7;
      PE_ID_I_L2 : Int := 8;
      PE_ID_I_L3 : Int := 9;
      PE_ID_S_L1 : Int := 10;
      PE_ID_S_L2 : Int := 11;
      PE_ID_S_L3 : Int := 12;
      PE_ID_P_L1 : Int := 13;
      PE_ID_P_L2 : Int := 14;
      PE_ID_P_L3 : Int := 15;
      PE_ID_Q_L1 : Int := 16;
      PE_ID_Q_L2 : Int := 17;
      PE_ID_Q_L3 : Int := 18;
      PE_ID_COS_L1 : Int := 19;
      PE_ID_COS_L2 : Int := 20;
      PE_ID_COS_L3 : Int := 21;
      PE_ID_F : Int := 22;
      PE_ID_U_AVG_L_N : Int := 23;
      PE_ID_U_AVG_L_L : Int := 24;
      PE_ID_I_AVG : Int := 25;
      PE_ID_P_OVERALL : Int := 26;
      PE_ID_Q_OVERALL : Int := 27;
      PE_ID_S_OVERALL : Int := 28;
      PE_ID_COS_OVERALL : Int := 29;
      PE_ID_U_L1_MAX : Int := 30;
      PE_ID_U_L2_MAX : Int := 31;
      PE_ID_U_L3_MAX : Int := 32;
      PE_ID_U_L1_L2_MAX : Int := 33;
      PE_ID_U_L2_L3_MAX : Int := 34;
      PE_ID_U_L3_L1_MAX : Int := 35;
      PE_ID_I_L1_MAX : Int := 36;
      PE_ID_I_L2_MAX : Int := 37;
      PE_ID_I_L3_MAX : Int := 38;
      PE_ID_S_L1_MAX : Int := 39;
      PE_ID_S_L2_MAX : Int := 40;
      PE_ID_S_L3_MAX : Int := 41;
      PE_ID_P_L1_MAX : Int := 42;
      PE_ID_P_L2_MAX : Int := 43;
      PE_ID_P_L3_MAX : Int := 44;
      PE_ID_Q_L1_MAX : Int := 45;
      PE_ID_Q_L2_MAX : Int := 46;
      PE_ID_Q_L3_MAX : Int := 47;
      PE_ID_COS_L1_MAX : Int := 48;
      PE_ID_COS_L2_MAX : Int := 49;
      PE_ID_COS_L3_MAX : Int := 50;
      PE_ID_F_MAX : Int := 51;
      PE_ID_U_AVG_L_N_MAX : Int := 52;
      PE_ID_U_AVG_L_L_MAX : Int := 53;
      PE_ID_I_AVG_MAX : Int := 54;
      PE_ID_P_OVERALL_MAX : Int := 55;
      PE_ID_Q_OVERALL_MAX : Int := 56;
      PE_ID_S_OVERALL_MAX : Int := 57;
      PE_ID_COS_OVERALL_MAX : Int := 58;
      PE_ID_U_L1_MIN : Int := 59;
      PE_ID_U_L2_MIN : Int := 60;
      PE_ID_U_L3_MIN : Int := 61;
      PE_ID_U_L1_L2_MIN : Int := 62;
      PE_ID_U_L2_L3_MIN : Int := 63;
      PE_ID_U_L3_L1_MIN : Int := 64;
      PE_ID_I_L1_MIN : Int := 65;
      PE_ID_I_L2_MIN : Int := 66;
      PE_ID_I_L3_MIN : Int := 67;
      PE_ID_S_L1_MIN : Int := 68;
      PE_ID_S_L2_MIN : Int := 69;
      PE_ID_S_L3_MIN : Int := 70;
      PE_ID_P_L1_MIN : Int := 71;
      PE_ID_P_L2_MIN : Int := 72;
      PE_ID_P_L3_MIN : Int := 73;
      PE_ID_Q_L1_MIN : Int := 74;
      PE_ID_Q_L2_MIN : Int := 75;
      PE_ID_Q_L3_MIN : Int := 76;
      PE_ID_COS_L1_MIN : Int := 77;
      PE_ID_COS_L2_MIN : Int := 78;
      PE_ID_COS_L3_MIN : Int := 79;
      PE_ID_F_MIN : Int := 80;
      PE_ID_U_AVG_L_N_MIN : Int := 81;
      PE_ID_U_AVG_L_L_MIN : Int := 82;
      PE_ID_I_AVG_MIN : Int := 83;
      PE_ID_P_OVERALL_MIN : Int := 84;
      PE_ID_Q_OVERALL_MIN : Int := 85;
      PE_ID_S_OVERALL_MIN : Int := 86;
      PE_ID_COS_OVERALL_MIN : Int := 87;
      PE_ID_E_P_IMP_64 : Int := 88;
      PE_ID_E_P_EXP_64 : Int := 89;
      PE_ID_E_Q_IMP_64 : Int := 90;
      PE_ID_E_Q_EXP_64 : Int := 91;
      PE_ID_E_S_IMP_64 : Int := 92;
   END_VAR
   // Receive_Data_Buffer[1..1000] := BYTE#16#00;
   // Send_Data_Buffer[1..240] := BYTE#16#00;
BEGIN



       // Only check the input variables during the first configuration or
       // until they are correct
       IF (#Input_Variables_OK = FALSE) THEN

           // Also check if a variable is connected to the communication
           // resource counter
           #In_Out_Pointer_Check := #Comm_Resource_Counter;

           // Check each input value for the correct value range
           // The ID of the Energy Meter has to be something bigger than 0
           // as the input bytes can't be negativ
           IF (#ID < 0) THEN

               // Set the error location and the error code for this error
               #Error_Location := #ERR_LOC_INVALID_ID;
               #Error_Code := #ERR_CODE_GENERAL;

               // The First_Byte_I_O_Data of the Energy Meter has to be something bigger than 0
               // as the input bytes can't be negativ
           ELSIF (#First_Byte_I_O_Data < 0) THEN

               // Set the error location and the error code for this error
               #Error_Location := #ERR_LOC_INVALID_IO_BYTE;
               #Error_Code := #ERR_CODE_GENERAL;

               // The available measurement types are only 1 phase measurement with
               // neutral (1), 3 phase measurement without neutral (3) and 3 phase
               // measurement with neutral (4)
           ELSIF ((#Connection_Type <> #CONNECTION_SINGLE_PHASE)
               AND (#Connection_Type <> #CONNECTION_THREE_PHASE)) THEN

               // Set the error location and the error code for this error
               #Error_Location := #ERR_LOC_INVALID_CONNECTION_TYPE;
               #Error_Code := #ERR_CODE_GENERAL;

               // The communication resource limit has to be somehting bigger than 0.
               // Otherwise, there will never be an update of the data
           ELSIF (#Comm_Resource_Limit <= 0) THEN

               // Set the error location and the error code for this error
               #Error_Location := #ERR_LOC_INVALID_COMM_LIMIT;
               #Error_Code := #ERR_CODE_GENERAL;

               // The available communication types are 1 (PROFINET) and 2 (PROFIBUS)
           ELSIF ((#Comm_Type <> #PROFINET)
               AND (#Comm_Type <> #PROFIBUS)) THEN

               // Set the error location and the error code for this error
               #Error_Location := #ERR_LOC_INVALID_COMM_TYPE;
               #Error_Code := #ERR_CODE_GENERAL;

               // A counter for the used resources has to be connected to work
               // If no variable is connected, the DB number and the DB offset
               // are both 0
           ELSIF (((#VIn_Out_Pointer_Check.DB_Number = 0)
               AND (#VIn_Out_Pointer_Check.DB_Offset = 0))
               OR ((#VIn_Out_Pointer_Check.ID_Type <> #DATA_TYPE_WORD)
               AND (#VIn_Out_Pointer_Check.ID_Type <> #DATA_TYPE_INT))
               OR (#VIn_Out_Pointer_Check.Count <> W#16#0001)) THEN

               // Set the error location and the error code for this error
               #Error_Location := #ERR_LOC_INVALID_COMM_COUNTER;
               #Error_Code := #ERR_CODE_GENERAL;

               // No error in the input variables
           ELSE

               // Check if a variable is connected to the HMI Input bits
               // If not, do not try to use these bits and only use internal
               // variables
               #In_Out_Pointer_Check := #HMI_Bits;

               // There is only nothing connected if the DB number is 0 
               // and the DB offset is also 0
               IF ((#VIn_Out_Pointer_Check.DB_Number = 0)
                   AND (#VIn_Out_Pointer_Check.DB_Offset = 0)) THEN

                   // Set the signal, that no structure is connected to the 
                   // HMI input bits
                   #HMI_Input_Bits_Connected := FALSE;
               ELSE
                   // A structure is connected and can be used in the program
                   #HMI_Input_Bits_Connected := TRUE;
               END_IF;

               // Set the signal, that all input variables are OK
               #Input_Variables_OK := TRUE;
           END_IF;

           // The input variables are checked and are OK
       ELSE

           // If a structure is connected to the HMI_Bits input structure
           // copy the values to the internal structure.
           // Otherwise use the initial values of the internal structure.
           IF (#HMI_Input_Bits_Connected = TRUE) THEN

               // Copy the variable to an internal structure
               #HMI_Bits_Internal := #HMI_Bits;
           ELSE
               ; // Use the initial values of the structure variables
           END_IF;

           // Call the instance of the SFB once at the beginning at the code and set its signal during the program
           #Read_Data_Record(REQ := #Read_Data_Rec_Request,
                             ID := #ID, //INT_TO_DWORD(#ID),
                             INDEX := #Rd_Rec_Index,
                             MLEN := #Rd_Rec_Max_Length,
                             RECORD := #Receive_Data_Buffer);

           // Call the instance of the SFB once at the beginning at the code and set its signal during the program
          #Write_Data_Record(REQ := #Write_Data_Rec_Request,
                             ID := #ID,//INT_TO_DWORD(#ID),
                             INDEX := #Wr_Rec_Index,
                             LEN := #Wr_Rec_Max_Length,
                             RECORD := #Send_Data_Buffer);

           // Keep the timer always running to get the time between two updates and during one update
           #Time_Measurement(IN := TRUE,
                             PT := T#21d);

           // Only call the the timer once at the beginning
           #Error_Retry_Timer(IN := #Error_Retry_Timer_Run,
                              PT := #TIME_RETRY_TIMER);

           // Only call the the timer once at the beginning
           #Watchdog(IN := #Watchdog_Run,
                     PT := #TIME_WATCHDOG);

           // Only call the the timer once at the beginning
           #Reset_Timer(IN := #Reset_Timer_Run,
                       PT := #TIME_RESET_TIMER);

           //===========================================================================
           //====== Set the values for the faceplate for E2M ===========================
           //===========================================================================

           // Set the values for the faceplate, to know which values should be displayed
           // First divide by the different measurement types, as different values
           // are activated in the faceplate for different measurement values
           CASE #Connection_Type OF

                   // 1 phase measurement with only L1 and neutral
               #CONNECTION_SINGLE_PHASE:

                   // The values are coded as bit arrays and can be checked in the manual
                   #Driver_Data.U_PH_N_Mod := W#16#1180;
                   #Driver_Data.U_PH_PH_Mod := W#16#0000;
                   #Driver_Data.I_Mod := W#16#1180;
                   #Driver_Data.S_Mod := W#16#1180;
                   #Driver_Data.P_Mod := W#16#1180;
                   #Driver_Data.Q_Mod := W#16#1180;
                   #Driver_Data.E_Mod := W#16#3381;
                   #Driver_Data.f_Mod := W#16#0380;
                   #Driver_Data.Cos_Mod := W#16#1180;

                   // 3 phase measurement with neutral
               #CONNECTION_THREE_PHASE:

                   // The values are coded as bit arrays and can be checked in the manual
                   #Driver_Data.U_PH_N_Mod := W#16#FF80;
                   #Driver_Data.U_PH_PH_Mod := W#16#FF80;
                   #Driver_Data.I_Mod := W#16#FF80;
                   #Driver_Data.S_Mod := W#16#FF80;
                   #Driver_Data.P_Mod := W#16#FF80;
                   #Driver_Data.Q_Mod := W#16#FF80;
                   #Driver_Data.E_Mod := W#16#3381;
                   #Driver_Data.f_Mod := W#16#0380;
                   #Driver_Data.Cos_Mod := W#16#FF80;

               ELSE
                   ; // Not possible, no other measurement type possible
           END_CASE;

           // Check if the minimum and maximum values are calculated or downloaded
           IF ((#Min_Max_Calculated = TRUE)
               AND (#Comm_Type = #PROFIBUS)) THEN

               // Set the signals, which values are calculated
               #Driver_Data.Calculate_Value1 := W#16#FF0F;
               #Driver_Data.Calculate_Value2 := W#16#F66F;
               #Driver_Data.Calculate_Value3 := W#16#B60D;
               #Driver_Data.Calculate_Value4 := W#16#B60D;
               #Driver_Data.Calculate_Value5 := W#16#B60D;
               #Driver_Data.Calculate_Value6 := W#16#BF07;
           ELSE

               // No value is calculated
               #Driver_Data.Calculate_Value1 := W#16#0000;
               #Driver_Data.Calculate_Value2 := W#16#0000;
               #Driver_Data.Calculate_Value3 := W#16#0000;
               #Driver_Data.Calculate_Value4 := W#16#0000;
               #Driver_Data.Calculate_Value5 := W#16#0000;
               #Driver_Data.Calculate_Value6 := W#16#0000;
           END_IF;

           //===========================================================================
           //====== Reset the minimum and maximum values ===============================
           //===========================================================================

           // With a request from the faceplate, reset all minimum and maximum values
           IF (((#HMI_Bits_Internal.Reset_min_max_Data = TRUE)
               AND (#Reset_Min_Max_HMI_Old = FALSE))
               OR ((#Reset_Min_Max = TRUE)
               AND (#Reset_Min_Max_Old = FALSE))) THEN

               // If the values should be calculated, simply reset the values in the code
               IF ((#Min_Max_Calculated = TRUE)
                   AND (#Comm_Type = 2)) THEN

                   // With a positive request, reset all min and max values which are stored
                   // Voltage between phase and neutral
                   #Driver_Data.U_L1_min := #Driver_Data.U_L1;
                   #Driver_Data.U_L1_max := #Driver_Data.U_L1;
                   #Driver_Data.U_L2_min := #Driver_Data.U_L2;
                   #Driver_Data.U_L2_max := #Driver_Data.U_L2;
                   #Driver_Data.U_L3_min := #Driver_Data.U_L3;
                   #Driver_Data.U_L3_max := #Driver_Data.U_L3;

                   // Voltage between phase and phase
                   #Driver_Data.U_L1_L2_min := #Driver_Data.U_L1_L2;
                   #Driver_Data.U_L1_L2_max := #Driver_Data.U_L1_L2;
                   #Driver_Data.U_L2_L3_min := #Driver_Data.U_L2_L3;
                   #Driver_Data.U_L2_L3_max := #Driver_Data.U_L2_L3;
                   #Driver_Data.U_L3_L1_min := #Driver_Data.U_L3_L1;
                   #Driver_Data.U_L3_L1_max := #Driver_Data.U_L3_L1;

                   // Average voltages for both
                   #Driver_Data.U_PH_N_Average_min := #Driver_Data.U_PH_N_Average;
                   #Driver_Data.U_PH_N_Average_max := #Driver_Data.U_PH_N_Average;
                   #Driver_Data.U_PH_PH_Average_min := #Driver_Data.U_PH_PH_Average;
                   #Driver_Data.U_PH_PH_Average_max := #Driver_Data.U_PH_PH_Average;

                   // Current values including average
                   #Driver_Data.I_L1_min := #Driver_Data.I_L1;
                   #Driver_Data.I_L1_max := #Driver_Data.I_L1;
                   #Driver_Data.I_L2_min := #Driver_Data.I_L2;
                   #Driver_Data.I_L2_max := #Driver_Data.I_L2;
                   #Driver_Data.I_L3_min := #Driver_Data.I_L3;
                   #Driver_Data.I_L3_max := #Driver_Data.I_L3;
                   #Driver_Data.I_Average_min := #Driver_Data.I_Average;
                   #Driver_Data.I_Average_max := #Driver_Data.I_Average;

                   // Net frequency
                   #Driver_Data.f_min := #Driver_Data.f;
                   #Driver_Data.f_max := #Driver_Data.f;

                   // Apparent power including overall
                   #Driver_Data.S_L1_min := #Driver_Data.S_L1;
                   #Driver_Data.S_L1_max := #Driver_Data.S_L1;
                   #Driver_Data.S_L2_min := #Driver_Data.S_L2;
                   #Driver_Data.S_L2_max := #Driver_Data.S_L2;
                   #Driver_Data.S_L3_min := #Driver_Data.S_L3;
                   #Driver_Data.S_L3_max := #Driver_Data.S_L3;
                   #Driver_Data.S_Total_min := #Driver_Data.S_Total;
                   #Driver_Data.S_Total_max := #Driver_Data.S_Total;

                   // Reactive power including overall
                   #Driver_Data.Q_L1_min := #Driver_Data.Q_L1;
                   #Driver_Data.Q_L1_max := #Driver_Data.Q_L1;
                   #Driver_Data.Q_L2_min := #Driver_Data.Q_L2;
                   #Driver_Data.Q_L2_max := #Driver_Data.Q_L2;
                   #Driver_Data.Q_L3_min := #Driver_Data.Q_L3;
                   #Driver_Data.Q_L3_max := #Driver_Data.Q_L3;
                   #Driver_Data.Q_Total_min := #Driver_Data.Q_Total;
                   #Driver_Data.Q_Total_max := #Driver_Data.Q_Total;

                   // Effective power including overall
                   #Driver_Data.P_L1_min := #Driver_Data.P_L1;
                   #Driver_Data.P_L1_max := #Driver_Data.P_L1;
                   #Driver_Data.P_L2_min := #Driver_Data.P_L2;
                   #Driver_Data.P_L2_max := #Driver_Data.P_L2;
                   #Driver_Data.P_L3_min := #Driver_Data.P_L3;
                   #Driver_Data.P_L3_max := #Driver_Data.P_L3;
                   #Driver_Data.P_Total_min := #Driver_Data.P_Total;
                   #Driver_Data.P_Total_max := #Driver_Data.P_Total;

                   // Power factor including overall
                   #Driver_Data.Cos_L1_min := #Driver_Data.Cos_L1;
                   #Driver_Data.Cos_L1_max := #Driver_Data.Cos_L1;
                   #Driver_Data.Cos_L2_min := #Driver_Data.Cos_L2;
                   #Driver_Data.Cos_L2_max := #Driver_Data.Cos_L2;
                   #Driver_Data.Cos_L3_min := #Driver_Data.Cos_L3;
                   #Driver_Data.Cos_L3_max := #Driver_Data.Cos_L3;
                   #Driver_Data.Cos_Total_min := #Driver_Data.Cos_Total;
                   #Driver_Data.Cos_Total_max := #Driver_Data.Cos_Total;

                   // Reset also the maximum time between two updates
                   #Time_Between_Update_Max := T#0s;

                   // Set the time, when the min and max values have been reseted
                   #General_Ret_Val := RD_SYS_T(OUT => #Driver_Data.RTime_Data_Value);
               ELSE

                   // Reset also the maximum time between two updates
                   #Time_Between_Update_Max := T#0s;

                   // Set the request to reset the minimum and maximum values
                   #Reset_Min_Max_Request := TRUE;
               END_IF;
           ELSE
               ; // No request for a reset
           END_IF;

           //===========================================================================
           //====== Check for a request to reset the energy counter ====================
           //===========================================================================

           // The energy counter reset can either be triggered from the input of
           // the driver or from the faceplate
           IF (((#Reset_Energy_Counter = TRUE)
               AND (#Reset_Energy_Old = FALSE))
               OR ((#HMI_Bits_Internal.Reset_Energy_Meter = TRUE)
               AND (#Reset_Energy_HMI_Old = FALSE))) THEN

               // Set the request to reset the energy counter
               #Reset_En_Count_Request := TRUE;
           ELSE
               ; // No request detected
           END_IF;

           // Reset the outputs for reseting min and max values in the PAC by using 1
           // As the PAC needs some time, to recognize the positive edge, the outputs can't be 
           // reset directly after setting them
           IF (#Reset_Timer.Q = TRUE) THEN

               // Reset the timer
               #Reset_Timer_Run := FALSE;

               // Reset all control outputs
               //Q[#First_Byte_I_O_Data, #BIT_RESET_MINIMUM_VALUES] := FALSE;
               //Q[#First_Byte_I_O_Data, #BIT_RESET_MAXIMUM_VALUES] := FALSE;
               //Q[#First_Byte_I_O_Data, #BIT_RESET_ENERGY_COUNTER] := FALSE;
               #Driver_Control := #Driver_Control AND 16#0007;
           ELSE
               ; // Timer not finished or not started
           END_IF;

           // Set the state for the state machine
           #Sm_State := #Sm_State_Next;

           //===========================================================================
           //====== Wait for a request to update values or restore energy counter ======
           //===========================================================================

           // Start the state machine for the real functionality of the block
           CASE #Sm_State OF

                   // Wait for the request to update the energy counter or the measurement values
               #SM_IDLE:

                   // Set the state of the block to "Waiting for a new request"
                   #Error_Location := #STATUS_IDLE;

                   // Check for a request to reset the minimum and maximum values
                   IF (#Reset_Min_Max_Request = TRUE) THEN

                       // Reset the request signal
                       #Reset_Min_Max_Request := FALSE;

                       // Read the current time to set the timestamp of the reset of the minimum and maximum values
                       #General_Ret_Val := RD_SYS_T(OUT => #Driver_Data.RTime_Data_Value);

                       // Set the signal to run the reset timer to reset the outputs later
                       #Reset_Timer_Run := TRUE;

                       // The min and max values can only be reset by using 1 with the control bytes
                       // Byte n.0 = reset the minimum values
                       // Byte n.1 = reset the maximum values
                       //Q[#First_Byte_I_O_Data, #BIT_RESET_MINIMUM_VALUES] := TRUE;
                       //Q[#First_Byte_I_O_Data, #BIT_RESET_MAXIMUM_VALUES] := TRUE;
                       #Driver_Control := #Driver_Control OR 16#0003;

                       // Check for a request to reset the energy counter
                   ELSIF (#Reset_En_Count_Request = TRUE) THEN

                       // Reset the request signal
                       #Reset_En_Count_Request := FALSE;

                       // Read the current time to set the timestamp of the reset of the energy counter
                       #General_Ret_Val := RD_SYS_T(OUT => #Driver_Data.RTime_Data_Energy);

                       // Set the signal to run the reset timer to reset the outputs later
                       #Reset_Timer_Run := TRUE;

                       // The energy counter can only be reset by using 1 with the control bytes
                       // Byte n.2 = reset the energy counter
                       //Q[#First_Byte_I_O_Data, #BIT_RESET_ENERGY_COUNTER] := TRUE;
                       #Driver_Control := #Driver_Control OR 16#0001;

                       // Check if the update timer is elapsed ==> then start to update the measurement values
                   ELSIF (((#Automatic_Update = TRUE)
                       OR (#HMI_Bits_Internal.Start_Auto = TRUE)
                       OR ((#HMI_Bits_Internal.Start_Acyclic = TRUE)
                       AND (#Start_Acyclic_HMI_Old = FALSE)))
                       AND (#Comm_Resource_Limit > 0)) THEN

                       // Check the communication type, for the different data record communication
                       // The communication should happen with 1 ==> PROFIenergy
                       IF (#Comm_Type = #PROFINET) THEN

                           // Increase the request reference
                           #PE_Request_Reference := INT_TO_BYTE(BYTE_TO_INT(#PE_Request_Reference) + 1);

                           // The request refence could not be 0
                           IF (#PE_Request_Reference = B#16#00) THEN
                               #PE_Request_Reference := B#16#01;
                           ELSE
                               ; // Request reference valid
                           END_IF;

                           // For the communication with 1, PROFIenergy is used to get the measurement values. Therefore, data record
                           // 0x80A0 is used. Now build this data record, first the Block header.
                           #V_PN_Measurement_Data_1.Block_Header.Block_Type := W#16#0800;
                           #V_PN_Measurement_Data_1.Block_Header.Block_Version := W#16#0100;

                           // Now build the header special for PROFIenergy
                           #V_PN_Measurement_Data_1.Request_Header.Service_Request_ID := #PN_REQUEST_ID_GET_MEASUREMENT_VALUES;
                           #V_PN_Measurement_Data_1.Request_Header.Request_Reference := #PE_Request_Reference;
                           #V_PN_Measurement_Data_1.Service_Header_Request.Modifier := B#16#02;
                           #V_PN_Measurement_Data_1.Service_Header_Request.Data_Struct_Identifier := B#16#01;

                           // Now build the request data
                           #V_PN_Measurement_Data_1.Service_Data_Request.Count_Meas_Values := INT_TO_BYTE(#RECORD_PE_COUNT_MEAS_1);
                           #V_PN_Measurement_Data_1.Service_Data_Request.Meas_Values[PE_ID_U_L1] := 1;
                           #V_PN_Measurement_Data_1.Service_Data_Request.Meas_Values[PE_ID_U_L2] := 2;
                           #V_PN_Measurement_Data_1.Service_Data_Request.Meas_Values[PE_ID_U_L3] := 3;
                           #V_PN_Measurement_Data_1.Service_Data_Request.Meas_Values[PE_ID_U_L1_L2] := 4;
                           #V_PN_Measurement_Data_1.Service_Data_Request.Meas_Values[PE_ID_U_L2_L3] := 5;
                           #V_PN_Measurement_Data_1.Service_Data_Request.Meas_Values[PE_ID_U_L3_L1] := 6;
                           #V_PN_Measurement_Data_1.Service_Data_Request.Meas_Values[PE_ID_I_L1] := 7;
                           #V_PN_Measurement_Data_1.Service_Data_Request.Meas_Values[PE_ID_I_L2] := 8;
                           #V_PN_Measurement_Data_1.Service_Data_Request.Meas_Values[PE_ID_I_L3] := 9;
                           #V_PN_Measurement_Data_1.Service_Data_Request.Meas_Values[PE_ID_S_L1] := 10;
                           #V_PN_Measurement_Data_1.Service_Data_Request.Meas_Values[PE_ID_S_L2] := 11;
                           #V_PN_Measurement_Data_1.Service_Data_Request.Meas_Values[PE_ID_S_L3] := 12;
                           #V_PN_Measurement_Data_1.Service_Data_Request.Meas_Values[PE_ID_P_L1] := 13;
                           #V_PN_Measurement_Data_1.Service_Data_Request.Meas_Values[PE_ID_P_L2] := 14;
                           #V_PN_Measurement_Data_1.Service_Data_Request.Meas_Values[PE_ID_P_L3] := 15;
                           #V_PN_Measurement_Data_1.Service_Data_Request.Meas_Values[PE_ID_Q_L1] := 16;
                           #V_PN_Measurement_Data_1.Service_Data_Request.Meas_Values[PE_ID_Q_L2] := 17;
                           #V_PN_Measurement_Data_1.Service_Data_Request.Meas_Values[PE_ID_Q_L3] := 18;
                           #V_PN_Measurement_Data_1.Service_Data_Request.Meas_Values[PE_ID_COS_L1] := 19;
                           #V_PN_Measurement_Data_1.Service_Data_Request.Meas_Values[PE_ID_COS_L2] := 20;
                           #V_PN_Measurement_Data_1.Service_Data_Request.Meas_Values[PE_ID_COS_L3] := 21;
                           #V_PN_Measurement_Data_1.Service_Data_Request.Meas_Values[PE_ID_F] := 30;
                           #V_PN_Measurement_Data_1.Service_Data_Request.Meas_Values[PE_ID_U_AVG_L_N] := 31;
                           #V_PN_Measurement_Data_1.Service_Data_Request.Meas_Values[PE_ID_U_AVG_L_L] := 32;
                           #V_PN_Measurement_Data_1.Service_Data_Request.Meas_Values[PE_ID_I_AVG] := 33;
                           #V_PN_Measurement_Data_1.Service_Data_Request.Meas_Values[PE_ID_P_OVERALL] := 34;
                           #V_PN_Measurement_Data_1.Service_Data_Request.Meas_Values[PE_ID_Q_OVERALL] := 35;
                           #V_PN_Measurement_Data_1.Service_Data_Request.Meas_Values[PE_ID_S_OVERALL] := 36;
                           #V_PN_Measurement_Data_1.Service_Data_Request.Meas_Values[PE_ID_COS_OVERALL] := 37;

                           // Get the maximum values
                           #V_PN_Measurement_Data_1.Service_Data_Request.Meas_Values[PE_ID_U_L1_MAX] := 40;
                           #V_PN_Measurement_Data_1.Service_Data_Request.Meas_Values[PE_ID_U_L2_MAX] := 41;
                           #V_PN_Measurement_Data_1.Service_Data_Request.Meas_Values[PE_ID_U_L3_MAX] := 42;
                           #V_PN_Measurement_Data_1.Service_Data_Request.Meas_Values[PE_ID_U_L1_L2_MAX] := 43;
                           #V_PN_Measurement_Data_1.Service_Data_Request.Meas_Values[PE_ID_U_L2_L3_MAX] := 44;
                           #V_PN_Measurement_Data_1.Service_Data_Request.Meas_Values[PE_ID_U_L3_L1_MAX] := 45;
                           #V_PN_Measurement_Data_1.Service_Data_Request.Meas_Values[PE_ID_I_L1_MAX] := 46;
                           #V_PN_Measurement_Data_1.Service_Data_Request.Meas_Values[PE_ID_I_L2_MAX] := 47;
                           #V_PN_Measurement_Data_1.Service_Data_Request.Meas_Values[PE_ID_I_L3_MAX] := 48;
                           #V_PN_Measurement_Data_1.Service_Data_Request.Meas_Values[PE_ID_S_L1_MAX] := 49;
                           #V_PN_Measurement_Data_1.Service_Data_Request.Meas_Values[PE_ID_S_L2_MAX] := 50;
                           #V_PN_Measurement_Data_1.Service_Data_Request.Meas_Values[PE_ID_S_L3_MAX] := 51;
                           #V_PN_Measurement_Data_1.Service_Data_Request.Meas_Values[PE_ID_P_L1_MAX] := 52;
                           #V_PN_Measurement_Data_1.Service_Data_Request.Meas_Values[PE_ID_P_L2_MAX] := 53;
                           #V_PN_Measurement_Data_1.Service_Data_Request.Meas_Values[PE_ID_P_L3_MAX] := 54;
                           #V_PN_Measurement_Data_1.Service_Data_Request.Meas_Values[PE_ID_Q_L1_MAX] := 55;
                           #V_PN_Measurement_Data_1.Service_Data_Request.Meas_Values[PE_ID_Q_L2_MAX] := 56;
                           #V_PN_Measurement_Data_1.Service_Data_Request.Meas_Values[PE_ID_Q_L3_MAX] := 57;
                           #V_PN_Measurement_Data_1.Service_Data_Request.Meas_Values[PE_ID_COS_L1_MAX] := 58;
                           #V_PN_Measurement_Data_1.Service_Data_Request.Meas_Values[PE_ID_COS_L2_MAX] := 59;
                           #V_PN_Measurement_Data_1.Service_Data_Request.Meas_Values[PE_ID_COS_L3_MAX] := 60;

                           // Configure the data record number and the length of the data record
                           #Wr_Rec_Index := WORD_TO_INT(#RECORD_PROFIENERGY_INDEX);
                           #Wr_Rec_Max_Length := #RECORD_PE_WRITE_LEN_1;
                           #V_PN_Measurement_Data_1.Block_Header.Block_Length := #Wr_Rec_Max_Length - 4;

                           // The PAC is connected with 2
                       ELSIF (#Comm_Type = 2) THEN

                           // Configure the data record to write the values to the SENTRON PAC, which should be provided in this data record
                           // As there are too many values which should be provided and the maximum length of the data record is 240 byte,
                           // the reading of the measurement values is divided into two cycles, if the min and max values should not be
                           // calculated in the FB

                           // In the first reading, get the current values from the SENTRON PAC.
                           // ==> Configure the data record, to get the values by using the block reading of more values with one command

                           // In the first block, read the voltage, current, apparent power, effective power, reactive power and the power factor
                           // The ID of the first measurement value to read is 1.
                           // 21 values will be read, length = 21*4 = 84 / 2 (unit is amount of words) = 42
                           #V_DP_Measurement_Data.Measurement_Data[1].Measurement_ID := 1;
                           #V_DP_Measurement_Data.Measurement_Data[1].Measurement_Len := 42;

                           // In the second block, read net frequency, the average values and the overall power values
                           // The ID of the first measurement value to read is 55.
                           // 8 values will be read, length = 8*4 = 32 / 2 (unit is amount of words) = 16
                           #V_DP_Measurement_Data.Measurement_Data[2].Measurement_ID := 55;
                           #V_DP_Measurement_Data.Measurement_Data[2].Measurement_Len := 16;

                           // In the third block, read all energy counter, which are neccessary
                           // The ID of the first measurement value to read is 801.
                           // 21 values will be read, length = 10*8 (LREAL) = 80 / 2 (unit is amount of words) = 40
                           #V_DP_Measurement_Data.Measurement_Data[3].Measurement_ID := 801;
                           #V_DP_Measurement_Data.Measurement_Data[3].Measurement_Len := 40;

                           // Configure the data record number and the length of the data record
                           #Wr_Rec_Index := #RECORD_47_FLEX_ACCESS_MEASUREMENT_INDEX;
                           #Wr_Rec_Max_Length := #RECORD_47_WRITE_MEASUREMENT_VALUES_LENGTH;
                       ELSE
                           ; // Further communication methods
                       END_IF;

                       // Check if currently a communication resource for the update is available
                       // otherwise go to a wait state to get a new free resource
                       IF (#Comm_Resource_Counter < #Comm_Resource_Limit) THEN

                           // Store the time between two updates
                           #Time_Between_Update := #Time_Measurement.ET;

                           // Check if the this is the maximum time between the updates
                           IF (#Time_Between_Update > #Time_Between_Update_Max) THEN

                               // Set the new maximum time
                               #Time_Between_Update_Max := #Time_Between_Update;
                           ELSE
                               ; // No new maximum detected
                           END_IF;

                           // Reset the timer to restart the time next time
                           #Time_Measurement(IN := FALSE,
                                             PT := T#21d);

                           // A new resource is used for the update for this block instance
                           // ==> increse the used resources by 1
                           #Comm_Resource_Counter := #Comm_Resource_Counter + 1;

                           // Start the writing of the configuration data
                           #Write_Data_Rec_Request := TRUE;

                           // Go to the state for waiting for the answer
                           #Sm_State_Next := #SM_WRITE_MEAS_WAIT_RESP;
                       ELSE

                           // Currently, no resource is available
                           // ==> Go to another state, to wait for a free resource
                           #Sm_State_Next := #SM_MEAS_WAIT_RESOURCE;
                       END_IF;
                   ELSE
                       ; // Timer not elapsed, Energy Meter connected an not request to reset counter
                   END_IF;

                   //===========================================================================
                   //====== Read measurement values ============================================
                   //===========================================================================

                   // Wait for a free communication resource on the CPU
               #SM_MEAS_WAIT_RESOURCE:

                   // Set the state of the block to "Waiting for a free ressource"
                   #Error_Location := #STATUS_WAIT_FOR_RESOURCE;

                   // Check if a resource is available
                   // ==> then start the request
                   IF (#Comm_Resource_Counter < #Comm_Resource_Limit) THEN

                       // A new resource is used for the update for this block instance
                       // ==> increse the used resources by 1
                       #Comm_Resource_Counter := #Comm_Resource_Counter + 1;

                       // Start the reading of the data record for the measurement values
                       #Write_Data_Rec_Request := TRUE;

                       // Store the time between two updates
                       #Time_Between_Update := #Time_Measurement.ET;

                       // Check if the this is the maximum time between the updates
                       IF (#Time_Between_Update > #Time_Between_Update_Max) THEN

                           // Set the new maximum time
                           #Time_Between_Update_Max := #Time_Between_Update;
                       ELSE
                           ; // No new maximum detected
                       END_IF;

                       // Reset the timer to restart the time next time
                       #Time_Measurement(IN := FALSE,
                                         PT := T#21d);

                       // Go to the state for waiting for the answer
                       #Sm_State_Next := #SM_WRITE_MEAS_WAIT_RESP;
                   ELSE
                       ; // Wait for a free resource
                   END_IF;

                   // Wait for the answer of the SENTRON PAC 4200
               #SM_WRITE_MEAS_WAIT_RESP:

                   // Set the state of the block to "Reading the measurement values"
                   #Error_Location := #STATUS_READ_MEAS;

                   // Start the watchdog, while waiting for a response
                   #Watchdog_Run := TRUE;

                   // The configuration of the data record 47 on the PAC 4200 failed with an error
                   IF ((#Write_Data_Record.ERROR = TRUE)
                       OR (#Watchdog.Q = TRUE)) THEN

                       // Reset the watchdog
                       #Watchdog_Run := FALSE;

                       // Save the error code for the user to display the error reason and location
                       #Error_Location := #ERR_LOC_WRITE_MEAS_1;
                       #Error_Code := #Write_Data_Record.STATUS;

                       // Reset the request bit to write a record to the Energy Meter for
                       // generating a positive edge with the next request
                       #Write_Data_Rec_Request := FALSE;

                       // Release the communication resource
                       #Comm_Resource_Counter := #Comm_Resource_Counter - 1;

                       // Go back to the main state and wait for a new request
                       #Sm_State_Next := #SM_IDLE;

                       // The configuration of the data record 47 on the PAC 4200 has been finished with success
                   ELSIF (#Write_Data_Record.DONE = TRUE) THEN

                       // Reset the watchdog
                       #Watchdog_Run := FALSE;

                       // Reset the error code and location
                       #Error_Code := DW#16#0000_0000;

                       // Reset the request bit to write a record to the SENTRON PAC 4200 for
                       // generating a positive edge with the next request
                       #Write_Data_Rec_Request := FALSE;

                       // Check the communication type, for the different data record communication
                       // The communication should happen with 1 ==> PROFIenergy
                       IF (#Comm_Type = #PROFINET) THEN

                           // Now configure the values to read these measurement values
                           #Rd_Rec_Index := WORD_TO_INT(#RECORD_PROFIENERGY_INDEX);
                           #Rd_Rec_Max_Length := #RECORD_PE_READ_LEN_1;

                           // The PAC is connected with 2
                       ELSIF (#Comm_Type = #PROFIBUS) THEN

                           // Now configure the values to read these measurement values
                           #Rd_Rec_Index := #RECORD_47_FLEX_ACCESS_MEASUREMENT_INDEX;
                           #Rd_Rec_Max_Length := #RECORD_47_READ_MEASUREMENT_VALUES_LENGTH;
                       ELSE
                           ; // Further communication methods
                       END_IF;

                       // Start the reading of the measurement values
                       #Read_Data_Rec_Request := TRUE;

                       // Go back to the main state and wait for a new request
                       #Sm_State_Next := #SM_READ_MEAS_WAIT_RESP;
                   ELSE
                       ; // Reading still in progress
                   END_IF;

                   // The wait state after an error
               #SM_READ_MEAS_WAIT_TIME:

                   // The timer has to run
                   #Error_Retry_Timer_Run := TRUE;

                   // If the timer elapsed, retry reading
                   IF (#Error_Retry_Timer.Q = TRUE) THEN

                       // Retry the reading
                       #Sm_State_Next := #SM_READ_MEAS_WAIT_RESP;
                   ELSE
                       ; // Still wait
                   END_IF;

                   // Wait for an answer of the reading of the current measuement values
               #SM_READ_MEAS_WAIT_RESP:

                   // Start the watchdog, while waiting for a response
                   #Watchdog_Run := TRUE;

                   // Set the request to true, if the bit is reset in case of an error
                   #Read_Data_Rec_Request := #Error_Retry_Timer.Q;

                   // The update of the data failed with an error
                   IF ((#Read_Data_Record.ERROR = TRUE)
                       OR (#Watchdog.Q = TRUE)) THEN

                       // Reset the request bit to read a record from the Energy Meter for
                       // generating a positive edge with the next request
                       #Read_Data_Rec_Request := FALSE;

                       // Increase the retries to get an answer
                       #Error_Retry_Counter := #Error_Retry_Counter + 1;

                       // Check if the device is still busy
                       IF (((#Read_Data_Record.STATUS = #ERROR_CODE_DEVICE_BUSY)
                           AND (#Error_Retry_Counter >= #ERROR_RETRY_LIMIT))
                           OR (#Read_Data_Record.STATUS <> #ERROR_CODE_DEVICE_BUSY)) THEN

                           // Reset the watchdog
                           #Watchdog_Run := FALSE;

                           // Save the time to update the values, even with an error
                           #Time_to_update := #Time_Measurement.ET;

                           // Reset the timer to restart the time next time
                           #Time_Measurement(IN := FALSE,
                                             PT := T#21d);

                           // Reset the timer
                           #Error_Retry_Timer_Run := FALSE;

                           // Reset the retry counter
                           #Error_Retry_Counter := 0;

                           // Save the error code for the user to display the error reason and location
                           #Error_Location := #ERR_LOC_READ_MEAS_1;
                           #Error_Code := #Read_Data_Record.STATUS;

                           // Release the communication resource
                           #Comm_Resource_Counter := #Comm_Resource_Counter - 1;

                           // Go back to the main state and wait for a new request
                           #Sm_State_Next := #SM_IDLE;
                       ELSE
                           // Reset the timer
                           #Error_Retry_Timer(IN := FALSE,
                                              PT := #TIME_RETRY_TIMER);

                           // Start the error timer
                           #Error_Retry_Timer_Run := TRUE;

                           // Go to the wait state
                           #Sm_State_Next := #SM_READ_MEAS_WAIT_TIME;
                       END_IF;

                       // The update of the has been finished with success
                   ELSIF (#Read_Data_Record.VALID = TRUE) THEN

                       // Reset the watchdog
                       #Watchdog_Run := FALSE;

                       // Reset the retry counter
                       #Error_Retry_Counter := 0;

                       // Reset the error code and location
                       #Error_Code := DW#16#0000_0000;

                       // Reset the request bit to read a record from the Energy Meter for
                       // generating a positive edge with the next request
                       #Read_Data_Rec_Request := FALSE;

                       // Check the communication type, for the different data record communication
                       // The communication should happen with 1 ==> PROFIenergy
                       IF (#Comm_Type = #PROFINET) THEN

                           // Check the header of the PROFIenergy response for an error
                           // First of all, check the block type for correctness, it must be W160801
                           IF (#V_PN_Meas_Data_Res_1.Block_Header.Block_Type <> #PN_BLOCK_TYPE_READ) THEN

                               // Set the error code and location
                               #Error_Location := #ERR_LOC_PN_INV_BLOCK_1;
                               #Error_Code := #ERR_CODE_GENERAL;

                               // Go back to the main state and wait for a new request
                               #Sm_State_Next := #SM_IDLE;

                               // Check the service request ID ==> it should be 0x10
                           ELSIF (#V_PN_Meas_Data_Res_1.Response_Header.Service_Request_ID <> #PN_REQUEST_ID_GET_MEASUREMENT_VALUES) THEN

                               // Set the error code and location
                               #Error_Location := #ERR_LOC_PN_INV_REQ_ID_1;
                               #Error_Code := #ERR_CODE_GENERAL;

                               // Go back to the main state and wait for a new request
                               #Sm_State_Next := #SM_IDLE;

                               // Check the request reference ==> should be the same as in the request
                           ELSIF (#V_PN_Meas_Data_Res_1.Response_Header.Request_Reference <> #PE_Request_Reference) THEN

                               // Set the error code and location
                               #Error_Location := #ERR_LOC_PN_INV_REQ_REF_1;
                               #Error_Code := #ERR_CODE_GENERAL;

                               // Go back to the main state and wait for a new request
                               #Sm_State_Next := #SM_IDLE;

                               // Check the status of the response ==> should be ready (0x01)
                           ELSIF (#V_PN_Meas_Data_Res_1.Service_Header_Response.Status <> B#16#01) THEN

                               // Set the error code and location
                               #Error_Location := #ERR_LOC_PN_PE_CMD_FAIL_1;
                               #Error_Code := #Read_Data_Record.STATUS;

                               // Go back to the main state and wait for a new request
                               #Sm_State_Next := #SM_IDLE;

                               // Check the data structure identifier ==> should be 0x01
                           ELSIF (#V_PN_Meas_Data_Res_1.Service_Header_Response.Data_Struct_Identifier <> B#16#01) THEN

                               // Set the error code and location
                               #Error_Location := #ERR_LOC_PN_INV_DATSTR_1;
                               #Error_Code := #ERR_CODE_GENERAL;

                               // Go back to the main state and wait for a new request
                               #Sm_State_Next := #SM_IDLE;

                               // The header is OK
                           ELSE

                               // The default value for a not measured value is DW16FFFF_FFFF
                               // ==> replace it with 0.0
                               // ==> Therefore check every value in a FOR-loop if it is the default value
                               FOR #Index := 1 TO #RECORD_PE_COUNT_MEAS_1 BY 1 DO
                                   IF (REAL_TO_DWORD(#V_PN_Meas_Data_Res_1.Service_Data_Response.Meas_Values_32Bit[#Index].Meas_Value) = DW#16#FFFF_FFFF) THEN
                                       #V_PN_Meas_Data_Res_1.Service_Data_Response.Meas_Values_32Bit[#Index].Meas_Value := 0.0;
                                   ELSE
                                       ; // Value is correct
                                   END_IF;
                               END_FOR;

                               // Copy the data to the output structure of the measurement values
                               // but only a view variables can be updated, cause only few of them
                               // are supported by the Energy Meter

                               // ================================================
                               // Proceed the voltage values for each phase
                               // ================================================
                               #Driver_Data.U_L1 := #V_PN_Meas_Data_Res_1.Service_Data_Response.Meas_Values_32Bit[PE_ID_U_L1].Meas_Value;
                               #Driver_Data.U_L2 := #V_PN_Meas_Data_Res_1.Service_Data_Response.Meas_Values_32Bit[PE_ID_U_L2].Meas_Value;
                               #Driver_Data.U_L3 := #V_PN_Meas_Data_Res_1.Service_Data_Response.Meas_Values_32Bit[PE_ID_U_L3].Meas_Value;
                               #Driver_Data.U_PH_N_Average := #V_PN_Meas_Data_Res_1.Service_Data_Response.Meas_Values_32Bit[PE_ID_U_AVG_L_N].Meas_Value;

                               // ================================================
                               // Proceed the voltage values for phase to phase
                               // ================================================
                               #Driver_Data.U_L1_L2 := #V_PN_Meas_Data_Res_1.Service_Data_Response.Meas_Values_32Bit[PE_ID_U_L1_L2].Meas_Value;
                               #Driver_Data.U_L2_L3 := #V_PN_Meas_Data_Res_1.Service_Data_Response.Meas_Values_32Bit[PE_ID_U_L2_L3].Meas_Value;
                               #Driver_Data.U_L3_L1 := #V_PN_Meas_Data_Res_1.Service_Data_Response.Meas_Values_32Bit[PE_ID_U_L3_L1].Meas_Value;
                               #Driver_Data.U_PH_PH_Average := #V_PN_Meas_Data_Res_1.Service_Data_Response.Meas_Values_32Bit[PE_ID_U_AVG_L_L].Meas_Value;

                               // ================================================
                               // Proceed the current for each phase
                               // ================================================
                               #Driver_Data.I_L1 := #V_PN_Meas_Data_Res_1.Service_Data_Response.Meas_Values_32Bit[PE_ID_I_L1].Meas_Value;
                               #Driver_Data.I_L2 := #V_PN_Meas_Data_Res_1.Service_Data_Response.Meas_Values_32Bit[PE_ID_I_L2].Meas_Value;
                               #Driver_Data.I_L3 := #V_PN_Meas_Data_Res_1.Service_Data_Response.Meas_Values_32Bit[PE_ID_I_L3].Meas_Value;
                               #Driver_Data.I_Average := #V_PN_Meas_Data_Res_1.Service_Data_Response.Meas_Values_32Bit[PE_ID_I_AVG].Meas_Value;

                               // ================================================
                               // Proceed the frequency for the complete net
                               // ================================================
                               #Driver_Data.f := #V_PN_Meas_Data_Res_1.Service_Data_Response.Meas_Values_32Bit[PE_ID_F].Meas_Value;

                               // ================================================
                               // Proceed the cos for each phase
                               // ================================================
                               #Driver_Data.Cos_L1 := #V_PN_Meas_Data_Res_1.Service_Data_Response.Meas_Values_32Bit[PE_ID_COS_L1].Meas_Value;
                               #Driver_Data.Cos_L2 := #V_PN_Meas_Data_Res_1.Service_Data_Response.Meas_Values_32Bit[PE_ID_COS_L2].Meas_Value;
                               #Driver_Data.Cos_L3 := #V_PN_Meas_Data_Res_1.Service_Data_Response.Meas_Values_32Bit[PE_ID_COS_L3].Meas_Value;
                               #Driver_Data.Cos_Total := #V_PN_Meas_Data_Res_1.Service_Data_Response.Meas_Values_32Bit[PE_ID_COS_OVERALL].Meas_Value;

                               // ================================================
                               // Proceed the apparent power for each phase
                               // ================================================
                               #Driver_Data.S_L1 := #V_PN_Meas_Data_Res_1.Service_Data_Response.Meas_Values_32Bit[PE_ID_S_L1].Meas_Value;
                               #Driver_Data.S_L2 := #V_PN_Meas_Data_Res_1.Service_Data_Response.Meas_Values_32Bit[PE_ID_S_L2].Meas_Value;
                               #Driver_Data.S_L3 := #V_PN_Meas_Data_Res_1.Service_Data_Response.Meas_Values_32Bit[PE_ID_S_L3].Meas_Value;
                               #Driver_Data.S_Total := #V_PN_Meas_Data_Res_1.Service_Data_Response.Meas_Values_32Bit[PE_ID_S_OVERALL].Meas_Value;

                               // ================================================
                               // Proceed the reactive power for each phase
                               // ================================================
                               #Driver_Data.Q_L1 := #V_PN_Meas_Data_Res_1.Service_Data_Response.Meas_Values_32Bit[PE_ID_Q_L1].Meas_Value;
                               #Driver_Data.Q_L2 := #V_PN_Meas_Data_Res_1.Service_Data_Response.Meas_Values_32Bit[PE_ID_Q_L2].Meas_Value;
                               #Driver_Data.Q_L3 := #V_PN_Meas_Data_Res_1.Service_Data_Response.Meas_Values_32Bit[PE_ID_Q_L3].Meas_Value;
                               #Driver_Data.Q_Total := #V_PN_Meas_Data_Res_1.Service_Data_Response.Meas_Values_32Bit[PE_ID_Q_OVERALL].Meas_Value;

                               // ================================================
                               // Proceed the effective power for each phase
                               // ================================================
                               #Driver_Data.P_L1 := #V_PN_Meas_Data_Res_1.Service_Data_Response.Meas_Values_32Bit[PE_ID_P_L1].Meas_Value;
                               #Driver_Data.P_L2 := #V_PN_Meas_Data_Res_1.Service_Data_Response.Meas_Values_32Bit[PE_ID_P_L2].Meas_Value;
                               #Driver_Data.P_L3 := #V_PN_Meas_Data_Res_1.Service_Data_Response.Meas_Values_32Bit[PE_ID_P_L3].Meas_Value;
                               #Driver_Data.P_Total := #V_PN_Meas_Data_Res_1.Service_Data_Response.Meas_Values_32Bit[PE_ID_P_OVERALL].Meas_Value;

                               //===========================================================================
                               //====== Generate the minimum and maximum values ============================
                               //===========================================================================

                               // ================================================
                               // Proceed the voltage values for each phase
                               // ================================================
                               #Driver_Data.U_L1_max := #V_PN_Meas_Data_Res_1.Service_Data_Response.Meas_Values_32Bit[PE_ID_U_L1_MAX].Meas_Value;
                               #Driver_Data.U_L2_max := #V_PN_Meas_Data_Res_1.Service_Data_Response.Meas_Values_32Bit[PE_ID_U_L2_MAX].Meas_Value;
                               #Driver_Data.U_L3_max := #V_PN_Meas_Data_Res_1.Service_Data_Response.Meas_Values_32Bit[PE_ID_U_L3_MAX].Meas_Value;
                               #Driver_Data.U_L1_L2_max := #V_PN_Meas_Data_Res_1.Service_Data_Response.Meas_Values_32Bit[PE_ID_U_L1_L2_MAX].Meas_Value;
                               #Driver_Data.U_L2_L3_max := #V_PN_Meas_Data_Res_1.Service_Data_Response.Meas_Values_32Bit[PE_ID_U_L2_L3_MAX].Meas_Value;
                               #Driver_Data.U_L3_L1_max := #V_PN_Meas_Data_Res_1.Service_Data_Response.Meas_Values_32Bit[PE_ID_U_L3_L1_MAX].Meas_Value;
                               #Driver_Data.I_L1_max := #V_PN_Meas_Data_Res_1.Service_Data_Response.Meas_Values_32Bit[PE_ID_I_L1_MAX].Meas_Value;
                               #Driver_Data.I_L2_max := #V_PN_Meas_Data_Res_1.Service_Data_Response.Meas_Values_32Bit[PE_ID_I_L2_MAX].Meas_Value;
                               #Driver_Data.I_L3_max := #V_PN_Meas_Data_Res_1.Service_Data_Response.Meas_Values_32Bit[PE_ID_I_L3_MAX].Meas_Value;
                               #Driver_Data.Cos_L1_max := #V_PN_Meas_Data_Res_1.Service_Data_Response.Meas_Values_32Bit[PE_ID_COS_L1_MAX].Meas_Value;
                               #Driver_Data.Cos_L2_max := #V_PN_Meas_Data_Res_1.Service_Data_Response.Meas_Values_32Bit[PE_ID_COS_L2_MAX].Meas_Value;
                               #Driver_Data.Cos_L3_max := #V_PN_Meas_Data_Res_1.Service_Data_Response.Meas_Values_32Bit[PE_ID_COS_L3_MAX].Meas_Value;
                               #Driver_Data.S_L1_max := #V_PN_Meas_Data_Res_1.Service_Data_Response.Meas_Values_32Bit[PE_ID_S_L1_MAX].Meas_Value;
                               #Driver_Data.S_L2_max := #V_PN_Meas_Data_Res_1.Service_Data_Response.Meas_Values_32Bit[PE_ID_S_L2_MAX].Meas_Value;
                               #Driver_Data.S_L3_max := #V_PN_Meas_Data_Res_1.Service_Data_Response.Meas_Values_32Bit[PE_ID_S_L3_MAX].Meas_Value;
                               #Driver_Data.Q_L1_max := #V_PN_Meas_Data_Res_1.Service_Data_Response.Meas_Values_32Bit[PE_ID_Q_L1_MAX].Meas_Value;
                               #Driver_Data.Q_L2_max := #V_PN_Meas_Data_Res_1.Service_Data_Response.Meas_Values_32Bit[PE_ID_Q_L2_MAX].Meas_Value;
                               #Driver_Data.Q_L3_max := #V_PN_Meas_Data_Res_1.Service_Data_Response.Meas_Values_32Bit[PE_ID_Q_L3_MAX].Meas_Value;
                               #Driver_Data.P_L1_max := #V_PN_Meas_Data_Res_1.Service_Data_Response.Meas_Values_32Bit[PE_ID_P_L1_MAX].Meas_Value;
                               #Driver_Data.P_L2_max := #V_PN_Meas_Data_Res_1.Service_Data_Response.Meas_Values_32Bit[PE_ID_P_L2_MAX].Meas_Value;
                               #Driver_Data.P_L3_max := #V_PN_Meas_Data_Res_1.Service_Data_Response.Meas_Values_32Bit[PE_ID_P_L3_MAX].Meas_Value;

                               // Preapre the data for the next write request
                               // Increase the request reference
                               #PE_Request_Reference := INT_TO_BYTE(BYTE_TO_INT(#PE_Request_Reference) + 1);

                               // The request refence could not be 0
                               IF (#PE_Request_Reference = B#16#00) THEN
                                   #PE_Request_Reference := B#16#01;
                               ELSE
                                   ; // Request reference valid
                               END_IF;

                               // For the communication with 1, PROFIenergy is used to get the measurement values. Therefore, data record
                               // 0x80A0 is used. Now build this data record, first the Block header.
                               #V_PN_Measurement_Data_2.Block_Header.Block_Type := W#16#0800;
                               #V_PN_Measurement_Data_2.Block_Header.Block_Version := W#16#0100;

                               // Now build the header special for PROFIenergy
                               #V_PN_Measurement_Data_2.Request_Header.Service_Request_ID := B#16#10;
                               #V_PN_Measurement_Data_2.Request_Header.Request_Reference := #PE_Request_Reference;
                               #V_PN_Measurement_Data_2.Service_Header_Request.Modifier := B#16#02;
                               #V_PN_Measurement_Data_2.Service_Header_Request.Data_Struct_Identifier := B#16#01;

